// TIA Portal V17 export
// export: Created 2023-02-14T02:49:47.3102049Z, ExportSetting WithDefaults, DisplayName Totally Integrated Automation Portal, DisplayVersion V17, DisplayName TIA Portal Openness, DisplayVersion V17, DisplayName TIA Portal Teamcenter Gateway, DisplayVersion V17, DisplayName TIA Portal Version Control Interface, DisplayVersion V17, DisplayName SINAMICS Startdrive Advanced, DisplayVersion V17, DisplayName SINAMICS Startdrive G130, G150, S120, S150, SINAMICS MV, S210, DisplayVersion V17, DisplayName SINAMICS Startdrive G110M, G120, G120C, G120D, G120P, G115D, DisplayVersion V17, DisplayName STEP 7 Professional, DisplayVersion V17, DisplayName STEP 7 Safety, DisplayVersion V17, DisplayName WinCC Professional, DisplayVersion V17
FUNCTION "Buffer" : Void   // FC11, LAD
{ S7_Optimized_Access := 'TRUE' }
VERSION : 0.1
// stored: AutoNumber true, IsIECCheckEnabled false, SetENOAutomatically false, UDAEnableTagReadback false
BEGIN

REGION Network 1: BFT 61 Rework 32
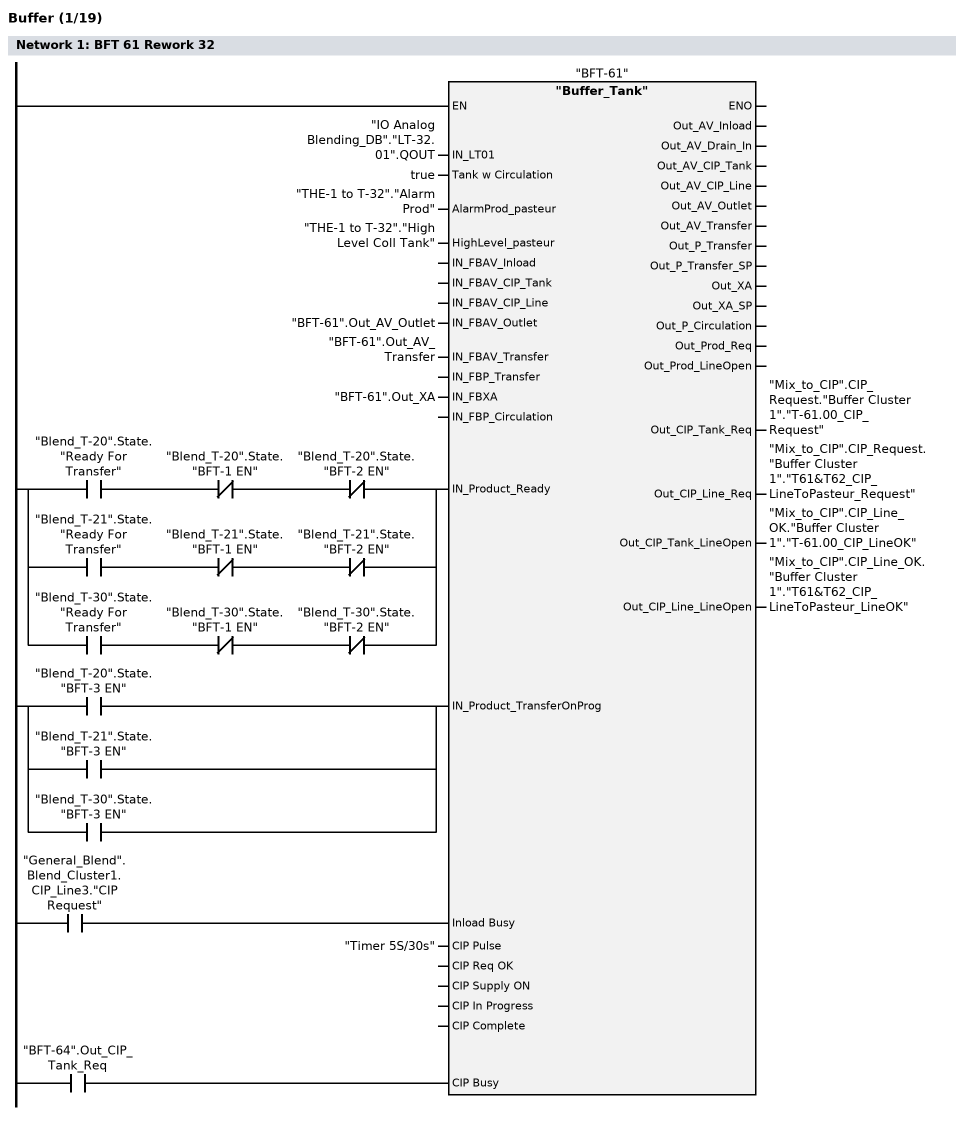
   RUNG wire#powerrail
      "BFT-61"(IN_Product_Ready := wire#w1, IN_Product_TransferOnProg := wire#w2, "Inload Busy" := wire#w3, "CIP Busy" := wire#w4, IN_LT01 := "IO Analog Blending_DB"."LT-32.01".QOUT, "Tank w Circulation" := true, AlarmProd_pasteur := "THE-1 to T-32"."Alarm Prod", HighLevel_pasteur := "THE-1 to T-32"."High Level Coll Tank", IN_FBAV_Inload :=, IN_FBAV_CIP_Tank :=, IN_FBAV_CIP_Line :=, IN_FBAV_Outlet := "BFT-61".Out_AV_Outlet, IN_FBAV_Transfer := "BFT-61".Out_AV_Transfer, IN_FBP_Transfer :=, IN_FBXA := "BFT-61".Out_XA, IN_FBP_Circulation :=, "CIP Pulse" := "Timer 5S/30s", "CIP Req OK" :=, "CIP Supply ON" :=, "CIP In Progress" :=, "CIP Complete" :=, Out_AV_Inload =>, Out_AV_Drain_In =>, Out_AV_CIP_Tank =>, Out_AV_CIP_Line =>, Out_AV_Outlet =>, Out_AV_Transfer =>, Out_P_Transfer =>, Out_P_Transfer_SP =>, Out_XA =>, Out_XA_SP =>, Out_P_Circulation =>, Out_Prod_Req =>, Out_Prod_LineOpen =>, Out_CIP_Tank_Req => "Mix_to_CIP".CIP_Request."Buffer Cluster 1"."T-61.00_CIP_Request", Out_CIP_Line_Req => "Mix_to_CIP".CIP_Request."Buffer Cluster 1"."T61&T62_CIP_LineToPasteur_Request", Out_CIP_Tank_LineOpen => "Mix_to_CIP".CIP_Line_OK."Buffer Cluster 1"."T-61.00_CIP_LineOK", Out_CIP_Line_LineOpen => "Mix_to_CIP".CIP_Line_OK."Buffer Cluster 1"."T61&T62_CIP_LineToPasteur_LineOK")
   END_RUNG
   RUNG wire#powerrail
      Contact( "Blend_T-20".State."Ready For Transfer" )
      I_Contact( "Blend_T-20".State."BFT-1 EN" )
      I_Contact( "Blend_T-20".State."BFT-2 EN" )
   END_RUNG wire#w1
   RUNG wire#powerrail
      Contact( "Blend_T-21".State."Ready For Transfer" )
      I_Contact( "Blend_T-21".State."BFT-1 EN" )
      I_Contact( "Blend_T-21".State."BFT-2 EN" )
   END_RUNG wire#w1
   RUNG wire#powerrail
      Contact( "Blend_T-30".State."Ready For Transfer" )
      I_Contact( "Blend_T-30".State."BFT-1 EN" )
      I_Contact( "Blend_T-30".State."BFT-2 EN" )
   END_RUNG wire#w1
   RUNG wire#powerrail
      Contact( "Blend_T-20".State."BFT-3 EN" )
   END_RUNG wire#w2
   RUNG wire#powerrail
      Contact( "Blend_T-21".State."BFT-3 EN" )
   END_RUNG wire#w2
   RUNG wire#powerrail
      Contact( "Blend_T-30".State."BFT-3 EN" )
   END_RUNG wire#w2
   RUNG wire#powerrail
      Contact( "General_Blend".Blend_Cluster1.CIP_Line3."CIP Request" )
   END_RUNG wire#w3
   RUNG wire#powerrail
      Contact( "BFT-64".Out_CIP_Tank_Req )
   END_RUNG wire#w4
   // the same network as SCL:
   "BFT-61"(IN_LT01 := "IO Analog Blending_DB"."LT-32.01".QOUT,   // "Buffer_Tank"
            "Tank w Circulation" := true,
            AlarmProd_pasteur := "THE-1 to T-32"."Alarm Prod",
            HighLevel_pasteur := "THE-1 to T-32"."High Level Coll Tank",
            IN_FBAV_Outlet := "BFT-61".Out_AV_Outlet,
            IN_FBAV_Transfer := "BFT-61".Out_AV_Transfer,
            IN_FBXA := "BFT-61".Out_XA,
            IN_Product_Ready := ("Blend_T-20".State."Ready For Transfer" AND NOT "Blend_T-20".State."BFT-1 EN" AND NOT "Blend_T-20".State."BFT-2 EN") OR ("Blend_T-21".State."Ready For Transfer" AND NOT "Blend_T-21".State."BFT-1 EN" AND NOT "Blend_T-21".State."BFT-2 EN") OR ("Blend_T-30".State."Ready For Transfer" AND NOT "Blend_T-30".State."BFT-1 EN" AND NOT "Blend_T-30".State."BFT-2 EN"),
            IN_Product_TransferOnProg := "Blend_T-20".State."BFT-3 EN" OR "Blend_T-21".State."BFT-3 EN" OR "Blend_T-30".State."BFT-3 EN",
            "Inload Busy" := "General_Blend".Blend_Cluster1.CIP_Line3."CIP Request",
            "CIP Pulse" := "Timer 5S/30s",
            "CIP Busy" := "BFT-64".Out_CIP_Tank_Req,
            Out_CIP_Tank_Req => "Mix_to_CIP".CIP_Request."Buffer Cluster 1"."T-61.00_CIP_Request",
            Out_CIP_Line_Req => "Mix_to_CIP".CIP_Request."Buffer Cluster 1"."T61&T62_CIP_LineToPasteur_Request",
            Out_CIP_Tank_LineOpen => "Mix_to_CIP".CIP_Line_OK."Buffer Cluster 1"."T-61.00_CIP_LineOK",
            Out_CIP_Line_LineOpen => "Mix_to_CIP".CIP_Line_OK."Buffer Cluster 1"."T61&T62_CIP_LineToPasteur_LineOK");
END_REGION

REGION Network 2: BFT 61 Feedback Instrument
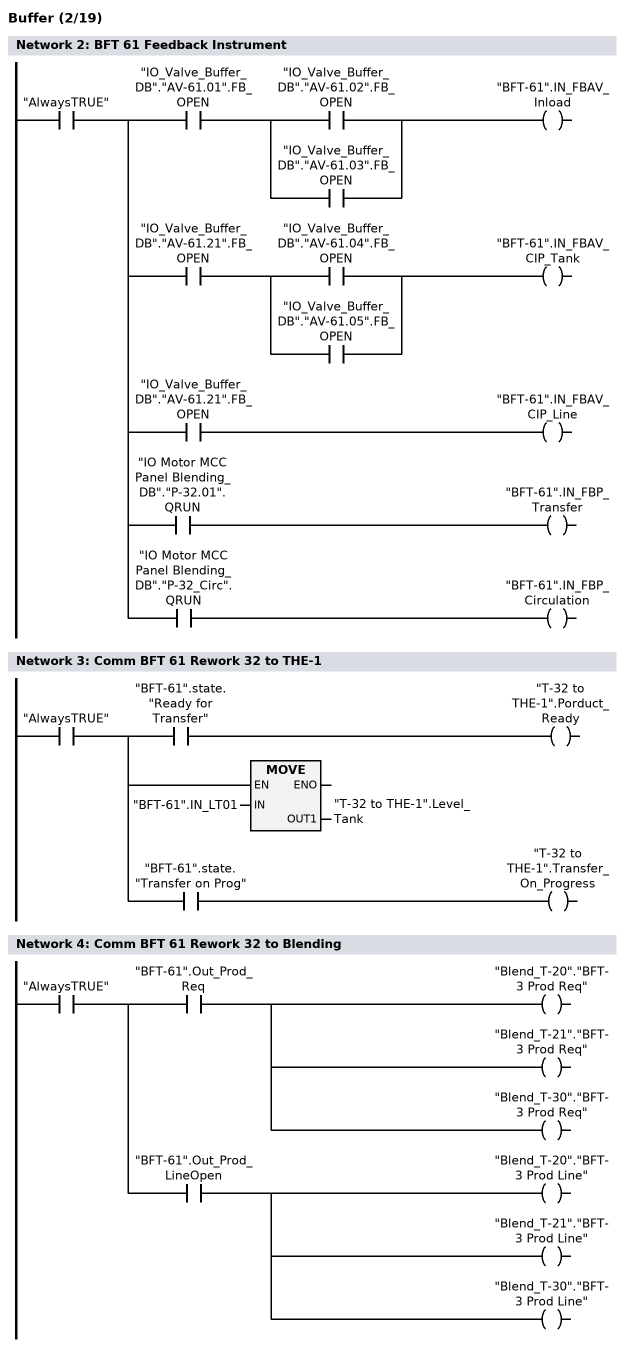
   RUNG wire#powerrail
      Contact( "AlwaysTRUE" )
      wire#w1
      Contact( "IO_Valve_Buffer_DB"."AV-61.01".FB_OPEN )
      wire#w2
      Contact( "IO_Valve_Buffer_DB"."AV-61.02".FB_OPEN )
      wire#w3
      Coil( "BFT-61".IN_FBAV_Inload )
   END_RUNG
   RUNG wire#w2
      Contact( "IO_Valve_Buffer_DB"."AV-61.03".FB_OPEN )
   END_RUNG wire#w3
   RUNG wire#w1
      Contact( "IO_Valve_Buffer_DB"."AV-61.21".FB_OPEN )
      wire#w4
      Contact( "IO_Valve_Buffer_DB"."AV-61.04".FB_OPEN )
      wire#w5
      Coil( "BFT-61".IN_FBAV_CIP_Tank )
   END_RUNG
   RUNG wire#w4
      Contact( "IO_Valve_Buffer_DB"."AV-61.05".FB_OPEN )
   END_RUNG wire#w5
   RUNG wire#w1
      Contact( "IO_Valve_Buffer_DB"."AV-61.21".FB_OPEN )
      Coil( "BFT-61".IN_FBAV_CIP_Line )
   END_RUNG
   RUNG wire#w1
      Contact( "IO Motor MCC Panel Blending_DB"."P-32.01".QRUN )
      Coil( "BFT-61".IN_FBP_Transfer )
   END_RUNG
   RUNG wire#w1
      Contact( "IO Motor MCC Panel Blending_DB"."P-32_Circ".QRUN )
      Coil( "BFT-61".IN_FBP_Circulation )
   END_RUNG
   // the same network as SCL:
   "BFT-61".IN_FBAV_Inload := "AlwaysTRUE" AND "IO_Valve_Buffer_DB"."AV-61.01".FB_OPEN AND ("IO_Valve_Buffer_DB"."AV-61.02".FB_OPEN OR "IO_Valve_Buffer_DB"."AV-61.03".FB_OPEN);
   "BFT-61".IN_FBAV_CIP_Tank := "AlwaysTRUE" AND "IO_Valve_Buffer_DB"."AV-61.21".FB_OPEN AND ("IO_Valve_Buffer_DB"."AV-61.04".FB_OPEN OR "IO_Valve_Buffer_DB"."AV-61.05".FB_OPEN);
   "BFT-61".IN_FBAV_CIP_Line := "AlwaysTRUE" AND "IO_Valve_Buffer_DB"."AV-61.21".FB_OPEN;
   "BFT-61".IN_FBP_Transfer := "AlwaysTRUE" AND "IO Motor MCC Panel Blending_DB"."P-32.01".QRUN;
   "BFT-61".IN_FBP_Circulation := "AlwaysTRUE" AND "IO Motor MCC Panel Blending_DB"."P-32_Circ".QRUN;
END_REGION

REGION Network 3: Comm BFT 61 Rework 32 to THE-1
   RUNG wire#powerrail
      Contact( "AlwaysTRUE" )
      wire#w1
      Contact( "BFT-61".state."Ready for Transfer" )
      Coil( "T-32 to THE-1".Porduct_Ready )
   END_RUNG
   RUNG wire#w1
      Move(in := "BFT-61".IN_LT01, out1 => "T-32 to THE-1".Level_Tank)
   END_RUNG
   RUNG wire#w1
      Contact( "BFT-61".state."Transfer on Prog" )
      Coil( "T-32 to THE-1".Transfer_On_Progress )
   END_RUNG
   // the same network as SCL:
   "T-32 to THE-1".Porduct_Ready := "AlwaysTRUE" AND "BFT-61".state."Ready for Transfer";
   IF "AlwaysTRUE" THEN "T-32 to THE-1".Level_Tank := "BFT-61".IN_LT01; END_IF;
   "T-32 to THE-1".Transfer_On_Progress := "AlwaysTRUE" AND "BFT-61".state."Transfer on Prog";
END_REGION

REGION Network 4: Comm BFT 61 Rework 32 to Blending
   RUNG wire#powerrail
      Contact( "AlwaysTRUE" )
      wire#w1
      Contact( "BFT-61".Out_Prod_Req )
      wire#w2
      Coil( "Blend_T-20"."BFT-3 Prod Req" )
   END_RUNG
   RUNG wire#w2
      Coil( "Blend_T-21"."BFT-3 Prod Req" )
   END_RUNG
   RUNG wire#w2
      Coil( "Blend_T-30"."BFT-3 Prod Req" )
   END_RUNG
   RUNG wire#w1
      Contact( "BFT-61".Out_Prod_LineOpen )
      wire#w3
      Coil( "Blend_T-20"."BFT-3 Prod Line" )
   END_RUNG
   RUNG wire#w3
      Coil( "Blend_T-21"."BFT-3 Prod Line" )
   END_RUNG
   RUNG wire#w3
      Coil( "Blend_T-30"."BFT-3 Prod Line" )
   END_RUNG
   // the same network as SCL:
   "Blend_T-20"."BFT-3 Prod Req" := "AlwaysTRUE" AND "BFT-61".Out_Prod_Req;
   "Blend_T-21"."BFT-3 Prod Req" := "Blend_T-20"."BFT-3 Prod Req";
   "Blend_T-30"."BFT-3 Prod Req" := "Blend_T-20"."BFT-3 Prod Req";
   "Blend_T-20"."BFT-3 Prod Line" := "AlwaysTRUE" AND "BFT-61".Out_Prod_LineOpen;
   "Blend_T-21"."BFT-3 Prod Line" := "Blend_T-20"."BFT-3 Prod Line";
   "Blend_T-30"."BFT-3 Prod Line" := "Blend_T-20"."BFT-3 Prod Line";
END_REGION

REGION Network 6: BFT 64 Rework 22
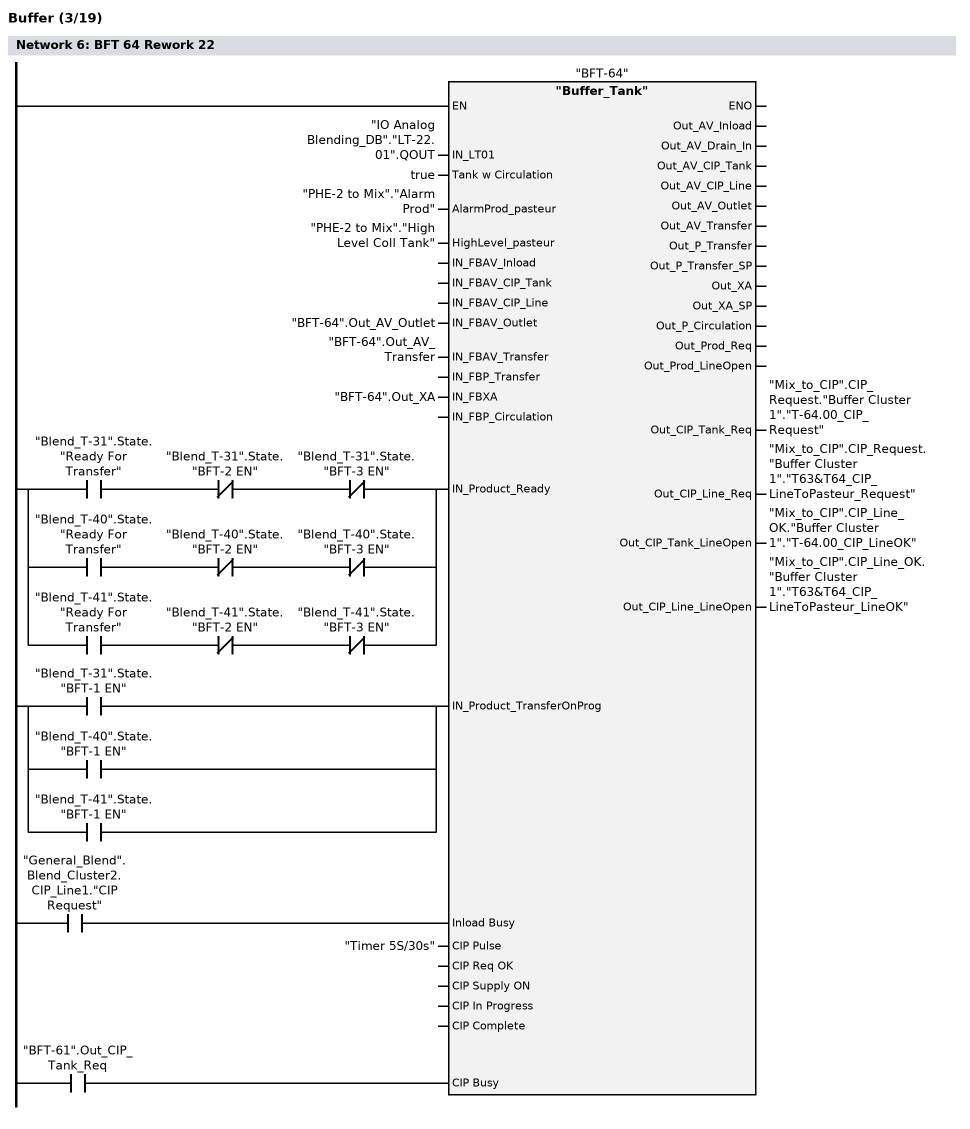
   RUNG wire#powerrail
      "BFT-64"(IN_Product_Ready := wire#w1, IN_Product_TransferOnProg := wire#w2, "Inload Busy" := wire#w3, "CIP Busy" := wire#w4, IN_LT01 := "IO Analog Blending_DB"."LT-22.01".QOUT, "Tank w Circulation" := true, AlarmProd_pasteur := "PHE-2 to Mix"."Alarm Prod", HighLevel_pasteur := "PHE-2 to Mix"."High Level Coll Tank", IN_FBAV_Inload :=, IN_FBAV_CIP_Tank :=, IN_FBAV_CIP_Line :=, IN_FBAV_Outlet := "BFT-64".Out_AV_Outlet, IN_FBAV_Transfer := "BFT-64".Out_AV_Transfer, IN_FBP_Transfer :=, IN_FBXA := "BFT-64".Out_XA, IN_FBP_Circulation :=, "CIP Pulse" := "Timer 5S/30s", "CIP Req OK" :=, "CIP Supply ON" :=, "CIP In Progress" :=, "CIP Complete" :=, Out_AV_Inload =>, Out_AV_Drain_In =>, Out_AV_CIP_Tank =>, Out_AV_CIP_Line =>, Out_AV_Outlet =>, Out_AV_Transfer =>, Out_P_Transfer =>, Out_P_Transfer_SP =>, Out_XA =>, Out_XA_SP =>, Out_P_Circulation =>, Out_Prod_Req =>, Out_Prod_LineOpen =>, Out_CIP_Tank_Req => "Mix_to_CIP".CIP_Request."Buffer Cluster 1"."T-64.00_CIP_Request", Out_CIP_Line_Req => "Mix_to_CIP".CIP_Request."Buffer Cluster 1"."T63&T64_CIP_LineToPasteur_Request", Out_CIP_Tank_LineOpen => "Mix_to_CIP".CIP_Line_OK."Buffer Cluster 1"."T-64.00_CIP_LineOK", Out_CIP_Line_LineOpen => "Mix_to_CIP".CIP_Line_OK."Buffer Cluster 1"."T63&T64_CIP_LineToPasteur_LineOK")
   END_RUNG
   RUNG wire#powerrail
      Contact( "Blend_T-31".State."Ready For Transfer" )
      I_Contact( "Blend_T-31".State."BFT-2 EN" )
      I_Contact( "Blend_T-31".State."BFT-3 EN" )
   END_RUNG wire#w1
   RUNG wire#powerrail
      Contact( "Blend_T-40".State."Ready For Transfer" )
      I_Contact( "Blend_T-40".State."BFT-2 EN" )
      I_Contact( "Blend_T-40".State."BFT-3 EN" )
   END_RUNG wire#w1
   RUNG wire#powerrail
      Contact( "Blend_T-41".State."Ready For Transfer" )
      I_Contact( "Blend_T-41".State."BFT-2 EN" )
      I_Contact( "Blend_T-41".State."BFT-3 EN" )
   END_RUNG wire#w1
   RUNG wire#powerrail
      Contact( "Blend_T-31".State."BFT-1 EN" )
   END_RUNG wire#w2
   RUNG wire#powerrail
      Contact( "Blend_T-40".State."BFT-1 EN" )
   END_RUNG wire#w2
   RUNG wire#powerrail
      Contact( "Blend_T-41".State."BFT-1 EN" )
   END_RUNG wire#w2
   RUNG wire#powerrail
      Contact( "General_Blend".Blend_Cluster2.CIP_Line1."CIP Request" )
   END_RUNG wire#w3
   RUNG wire#powerrail
      Contact( "BFT-61".Out_CIP_Tank_Req )
   END_RUNG wire#w4
   // the same network as SCL:
   "BFT-64"(IN_LT01 := "IO Analog Blending_DB"."LT-22.01".QOUT,   // "Buffer_Tank"
            "Tank w Circulation" := true,
            AlarmProd_pasteur := "PHE-2 to Mix"."Alarm Prod",
            HighLevel_pasteur := "PHE-2 to Mix"."High Level Coll Tank",
            IN_FBAV_Outlet := "BFT-64".Out_AV_Outlet,
            IN_FBAV_Transfer := "BFT-64".Out_AV_Transfer,
            IN_FBXA := "BFT-64".Out_XA,
            IN_Product_Ready := ("Blend_T-31".State."Ready For Transfer" AND NOT "Blend_T-31".State."BFT-2 EN" AND NOT "Blend_T-31".State."BFT-3 EN") OR ("Blend_T-40".State."Ready For Transfer" AND NOT "Blend_T-40".State."BFT-2 EN" AND NOT "Blend_T-40".State."BFT-3 EN") OR ("Blend_T-41".State."Ready For Transfer" AND NOT "Blend_T-41".State."BFT-2 EN" AND NOT "Blend_T-41".State."BFT-3 EN"),
            IN_Product_TransferOnProg := "Blend_T-31".State."BFT-1 EN" OR "Blend_T-40".State."BFT-1 EN" OR "Blend_T-41".State."BFT-1 EN",
            "Inload Busy" := "General_Blend".Blend_Cluster2.CIP_Line1."CIP Request",
            "CIP Pulse" := "Timer 5S/30s",
            "CIP Busy" := "BFT-61".Out_CIP_Tank_Req,
            Out_CIP_Tank_Req => "Mix_to_CIP".CIP_Request."Buffer Cluster 1"."T-64.00_CIP_Request",
            Out_CIP_Line_Req => "Mix_to_CIP".CIP_Request."Buffer Cluster 1"."T63&T64_CIP_LineToPasteur_Request",
            Out_CIP_Tank_LineOpen => "Mix_to_CIP".CIP_Line_OK."Buffer Cluster 1"."T-64.00_CIP_LineOK",
            Out_CIP_Line_LineOpen => "Mix_to_CIP".CIP_Line_OK."Buffer Cluster 1"."T63&T64_CIP_LineToPasteur_LineOK");
END_REGION

REGION Network 7: BFT 64 Feedback Instrument
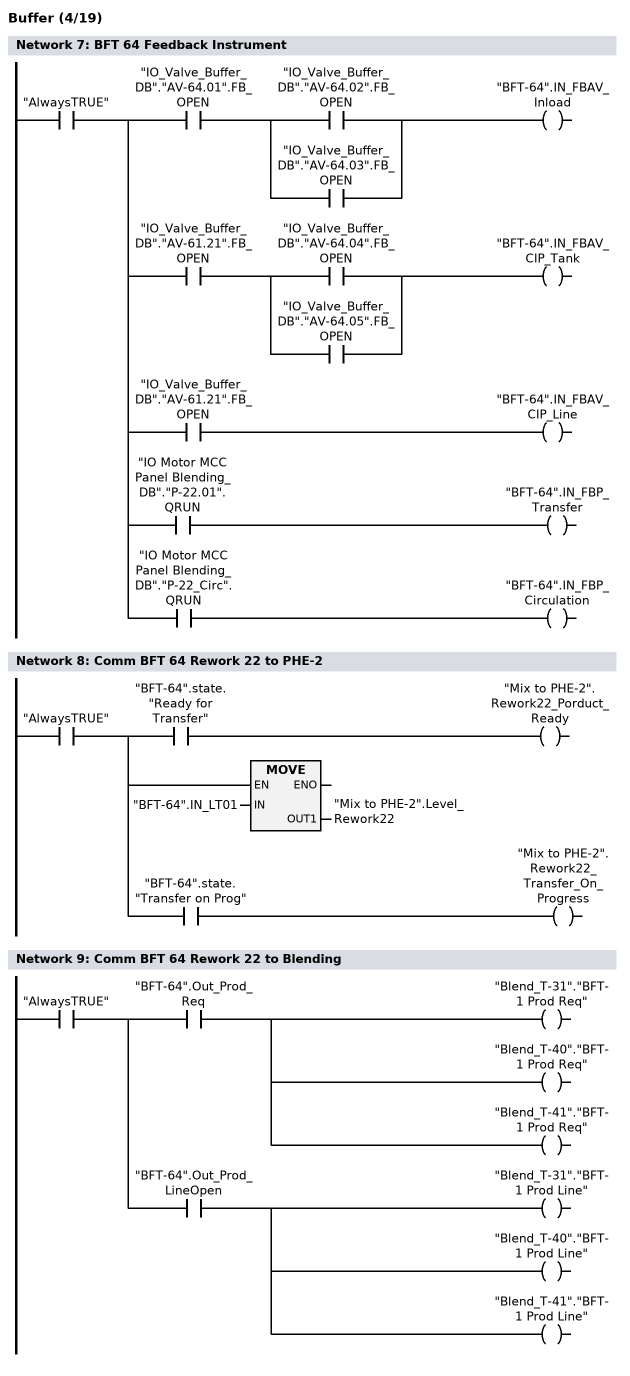
   RUNG wire#powerrail
      Contact( "AlwaysTRUE" )
      wire#w1
      Contact( "IO_Valve_Buffer_DB"."AV-64.01".FB_OPEN )
      wire#w2
      Contact( "IO_Valve_Buffer_DB"."AV-64.02".FB_OPEN )
      wire#w3
      Coil( "BFT-64".IN_FBAV_Inload )
   END_RUNG
   RUNG wire#w2
      Contact( "IO_Valve_Buffer_DB"."AV-64.03".FB_OPEN )
   END_RUNG wire#w3
   RUNG wire#w1
      Contact( "IO_Valve_Buffer_DB"."AV-61.21".FB_OPEN )
      wire#w4
      Contact( "IO_Valve_Buffer_DB"."AV-64.04".FB_OPEN )
      wire#w5
      Coil( "BFT-64".IN_FBAV_CIP_Tank )
   END_RUNG
   RUNG wire#w4
      Contact( "IO_Valve_Buffer_DB"."AV-64.05".FB_OPEN )
   END_RUNG wire#w5
   RUNG wire#w1
      Contact( "IO_Valve_Buffer_DB"."AV-61.21".FB_OPEN )
      Coil( "BFT-64".IN_FBAV_CIP_Line )
   END_RUNG
   RUNG wire#w1
      Contact( "IO Motor MCC Panel Blending_DB"."P-22.01".QRUN )
      Coil( "BFT-64".IN_FBP_Transfer )
   END_RUNG
   RUNG wire#w1
      Contact( "IO Motor MCC Panel Blending_DB"."P-22_Circ".QRUN )
      Coil( "BFT-64".IN_FBP_Circulation )
   END_RUNG
   // the same network as SCL:
   "BFT-64".IN_FBAV_Inload := "AlwaysTRUE" AND "IO_Valve_Buffer_DB"."AV-64.01".FB_OPEN AND ("IO_Valve_Buffer_DB"."AV-64.02".FB_OPEN OR "IO_Valve_Buffer_DB"."AV-64.03".FB_OPEN);
   "BFT-64".IN_FBAV_CIP_Tank := "AlwaysTRUE" AND "IO_Valve_Buffer_DB"."AV-61.21".FB_OPEN AND ("IO_Valve_Buffer_DB"."AV-64.04".FB_OPEN OR "IO_Valve_Buffer_DB"."AV-64.05".FB_OPEN);
   "BFT-64".IN_FBAV_CIP_Line := "AlwaysTRUE" AND "IO_Valve_Buffer_DB"."AV-61.21".FB_OPEN;
   "BFT-64".IN_FBP_Transfer := "AlwaysTRUE" AND "IO Motor MCC Panel Blending_DB"."P-22.01".QRUN;
   "BFT-64".IN_FBP_Circulation := "AlwaysTRUE" AND "IO Motor MCC Panel Blending_DB"."P-22_Circ".QRUN;
END_REGION

REGION Network 8: Comm BFT 64 Rework 22 to PHE-2
   RUNG wire#powerrail
      Contact( "AlwaysTRUE" )
      wire#w1
      Contact( "BFT-64".state."Ready for Transfer" )
      Coil( "Mix to PHE-2".Rework22_Porduct_Ready )
   END_RUNG
   RUNG wire#w1
      Move(in := "BFT-64".IN_LT01, out1 => "Mix to PHE-2".Level_Rework22)
   END_RUNG
   RUNG wire#w1
      Contact( "BFT-64".state."Transfer on Prog" )
      Coil( "Mix to PHE-2".Rework22_Transfer_On_Progress )
   END_RUNG
   // the same network as SCL:
   "Mix to PHE-2".Rework22_Porduct_Ready := "AlwaysTRUE" AND "BFT-64".state."Ready for Transfer";
   IF "AlwaysTRUE" THEN "Mix to PHE-2".Level_Rework22 := "BFT-64".IN_LT01; END_IF;
   "Mix to PHE-2".Rework22_Transfer_On_Progress := "AlwaysTRUE" AND "BFT-64".state."Transfer on Prog";
END_REGION

REGION Network 9: Comm BFT 64 Rework 22 to Blending
   RUNG wire#powerrail
      Contact( "AlwaysTRUE" )
      wire#w1
      Contact( "BFT-64".Out_Prod_Req )
      wire#w2
      Coil( "Blend_T-31"."BFT-1 Prod Req" )
   END_RUNG
   RUNG wire#w2
      Coil( "Blend_T-40"."BFT-1 Prod Req" )
   END_RUNG
   RUNG wire#w2
      Coil( "Blend_T-41"."BFT-1 Prod Req" )
   END_RUNG
   RUNG wire#w1
      Contact( "BFT-64".Out_Prod_LineOpen )
      wire#w3
      Coil( "Blend_T-31"."BFT-1 Prod Line" )
   END_RUNG
   RUNG wire#w3
      Coil( "Blend_T-40"."BFT-1 Prod Line" )
   END_RUNG
   RUNG wire#w3
      Coil( "Blend_T-41"."BFT-1 Prod Line" )
   END_RUNG
   // the same network as SCL:
   "Blend_T-31"."BFT-1 Prod Req" := "AlwaysTRUE" AND "BFT-64".Out_Prod_Req;
   "Blend_T-40"."BFT-1 Prod Req" := "Blend_T-31"."BFT-1 Prod Req";
   "Blend_T-41"."BFT-1 Prod Req" := "Blend_T-31"."BFT-1 Prod Req";
   "Blend_T-31"."BFT-1 Prod Line" := "AlwaysTRUE" AND "BFT-64".Out_Prod_LineOpen;
   "Blend_T-40"."BFT-1 Prod Line" := "Blend_T-31"."BFT-1 Prod Line";
   "Blend_T-41"."BFT-1 Prod Line" := "Blend_T-31"."BFT-1 Prod Line";
END_REGION

REGION Network 11: BFT 65
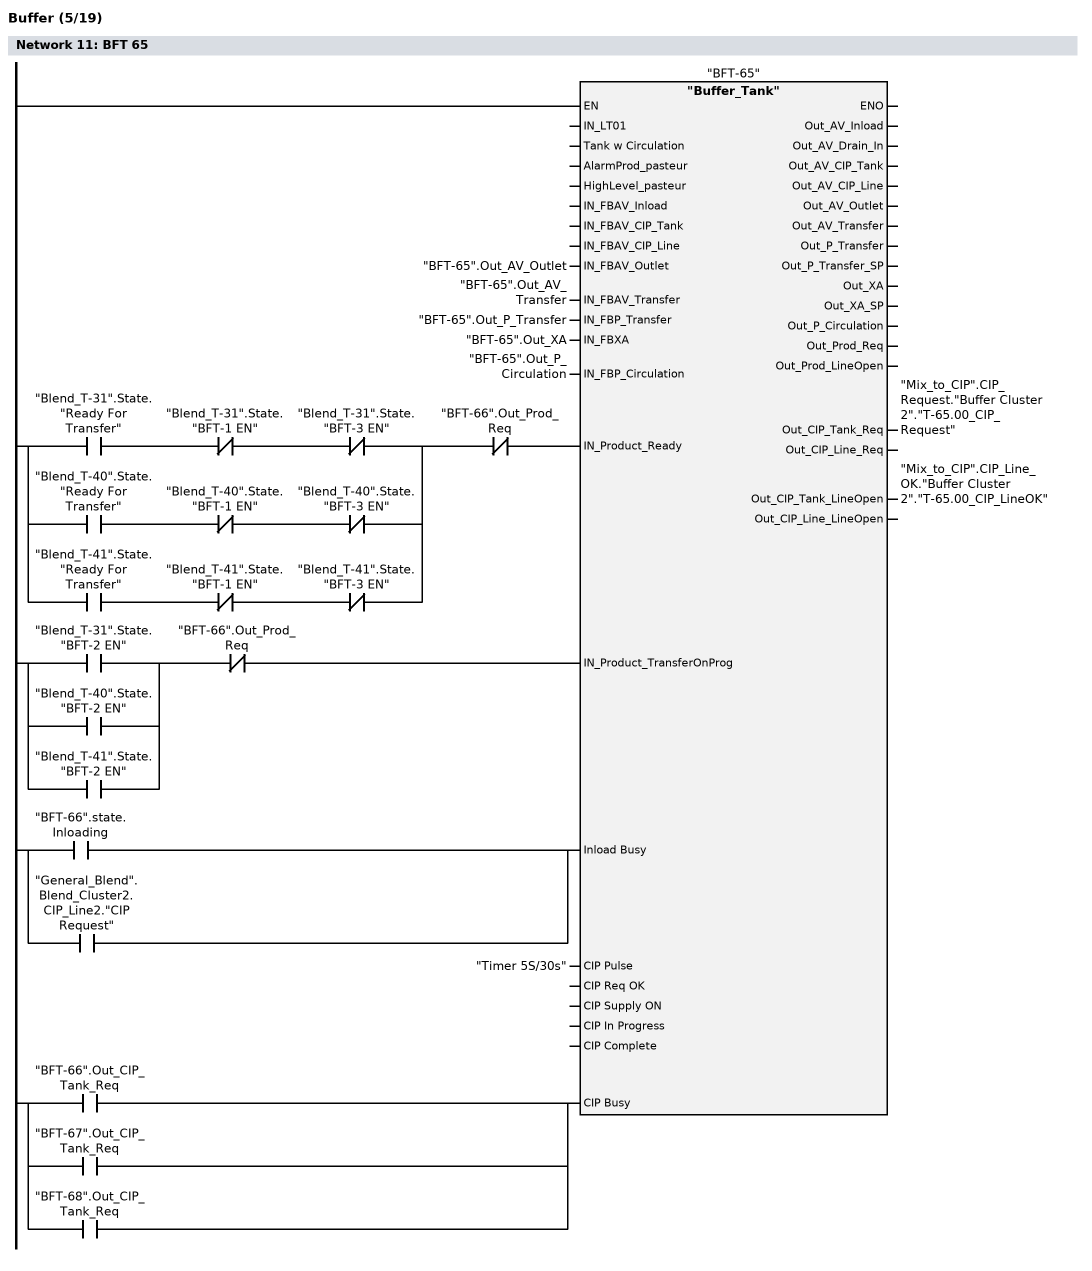
   RUNG wire#powerrail
      "BFT-65"(IN_Product_Ready := wire#w2, IN_Product_TransferOnProg := wire#w4, "Inload Busy" := wire#w5, "CIP Busy" := wire#w6, IN_LT01 :=, "Tank w Circulation" :=, AlarmProd_pasteur :=, HighLevel_pasteur :=, IN_FBAV_Inload :=, IN_FBAV_CIP_Tank :=, IN_FBAV_CIP_Line :=, IN_FBAV_Outlet := "BFT-65".Out_AV_Outlet, IN_FBAV_Transfer := "BFT-65".Out_AV_Transfer, IN_FBP_Transfer := "BFT-65".Out_P_Transfer, IN_FBXA := "BFT-65".Out_XA, IN_FBP_Circulation := "BFT-65".Out_P_Circulation, "CIP Pulse" := "Timer 5S/30s", "CIP Req OK" :=, "CIP Supply ON" :=, "CIP In Progress" :=, "CIP Complete" :=, Out_AV_Inload =>, Out_AV_Drain_In =>, Out_AV_CIP_Tank =>, Out_AV_CIP_Line =>, Out_AV_Outlet =>, Out_AV_Transfer =>, Out_P_Transfer =>, Out_P_Transfer_SP =>, Out_XA =>, Out_XA_SP =>, Out_P_Circulation =>, Out_Prod_Req =>, Out_Prod_LineOpen =>, Out_CIP_Tank_Req => "Mix_to_CIP".CIP_Request."Buffer Cluster 2"."T-65.00_CIP_Request", Out_CIP_Line_Req =>, Out_CIP_Tank_LineOpen => "Mix_to_CIP".CIP_Line_OK."Buffer Cluster 2"."T-65.00_CIP_LineOK", Out_CIP_Line_LineOpen =>)
   END_RUNG
   RUNG wire#powerrail
      Contact( "Blend_T-31".State."Ready For Transfer" )
      I_Contact( "Blend_T-31".State."BFT-1 EN" )
      I_Contact( "Blend_T-31".State."BFT-3 EN" )
      wire#w1
      I_Contact( "BFT-66".Out_Prod_Req )
   END_RUNG wire#w2
   RUNG wire#powerrail
      Contact( "Blend_T-40".State."Ready For Transfer" )
      I_Contact( "Blend_T-40".State."BFT-1 EN" )
      I_Contact( "Blend_T-40".State."BFT-3 EN" )
   END_RUNG wire#w1
   RUNG wire#powerrail
      Contact( "Blend_T-41".State."Ready For Transfer" )
      I_Contact( "Blend_T-41".State."BFT-1 EN" )
      I_Contact( "Blend_T-41".State."BFT-3 EN" )
   END_RUNG wire#w1
   RUNG wire#powerrail
      Contact( "Blend_T-31".State."BFT-2 EN" )
      wire#w3
      I_Contact( "BFT-66".Out_Prod_Req )
   END_RUNG wire#w4
   RUNG wire#powerrail
      Contact( "Blend_T-40".State."BFT-2 EN" )
   END_RUNG wire#w3
   RUNG wire#powerrail
      Contact( "Blend_T-41".State."BFT-2 EN" )
   END_RUNG wire#w3
   RUNG wire#powerrail
      Contact( "BFT-66".state.Inloading )
   END_RUNG wire#w5
   RUNG wire#powerrail
      Contact( "General_Blend".Blend_Cluster2.CIP_Line2."CIP Request" )
   END_RUNG wire#w5
   RUNG wire#powerrail
      Contact( "BFT-66".Out_CIP_Tank_Req )
   END_RUNG wire#w6
   RUNG wire#powerrail
      Contact( "BFT-67".Out_CIP_Tank_Req )
   END_RUNG wire#w6
   RUNG wire#powerrail
      Contact( "BFT-68".Out_CIP_Tank_Req )
   END_RUNG wire#w6
   // the same network as SCL:
   "BFT-65"(IN_FBAV_Outlet := "BFT-65".Out_AV_Outlet,   // "Buffer_Tank"
            IN_FBAV_Transfer := "BFT-65".Out_AV_Transfer,
            IN_FBP_Transfer := "BFT-65".Out_P_Transfer,
            IN_FBXA := "BFT-65".Out_XA,
            IN_FBP_Circulation := "BFT-65".Out_P_Circulation,
            IN_Product_Ready := (("Blend_T-31".State."Ready For Transfer" AND NOT "Blend_T-31".State."BFT-1 EN" AND NOT "Blend_T-31".State."BFT-3 EN") OR ("Blend_T-40".State."Ready For Transfer" AND NOT "Blend_T-40".State."BFT-1 EN" AND NOT "Blend_T-40".State."BFT-3 EN") OR ("Blend_T-41".State."Ready For Transfer" AND NOT "Blend_T-41".State."BFT-1 EN" AND NOT "Blend_T-41".State."BFT-3 EN")) AND NOT "BFT-66".Out_Prod_Req,
            IN_Product_TransferOnProg := ("Blend_T-31".State."BFT-2 EN" OR "Blend_T-40".State."BFT-2 EN" OR "Blend_T-41".State."BFT-2 EN") AND NOT "BFT-66".Out_Prod_Req,
            "Inload Busy" := "BFT-66".state.Inloading OR "General_Blend".Blend_Cluster2.CIP_Line2."CIP Request",
            "CIP Pulse" := "Timer 5S/30s",
            "CIP Busy" := "BFT-66".Out_CIP_Tank_Req OR "BFT-67".Out_CIP_Tank_Req OR "BFT-68".Out_CIP_Tank_Req,
            Out_CIP_Tank_Req => "Mix_to_CIP".CIP_Request."Buffer Cluster 2"."T-65.00_CIP_Request",
            Out_CIP_Tank_LineOpen => "Mix_to_CIP".CIP_Line_OK."Buffer Cluster 2"."T-65.00_CIP_LineOK");
END_REGION

REGION Network 12: BFT 65 Feedback Instrument
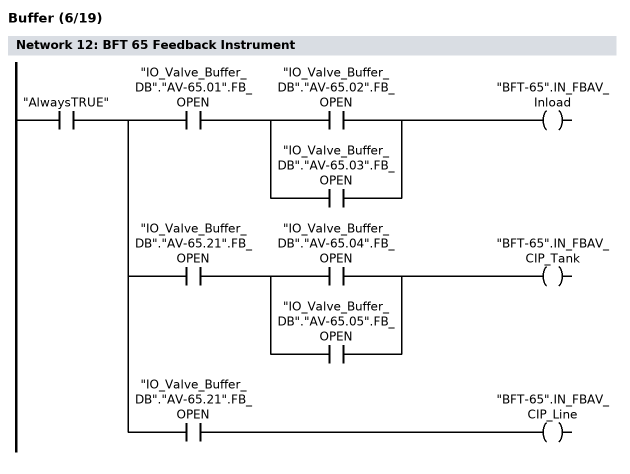
   RUNG wire#powerrail
      Contact( "AlwaysTRUE" )
      wire#w1
      Contact( "IO_Valve_Buffer_DB"."AV-65.01".FB_OPEN )
      wire#w2
      Contact( "IO_Valve_Buffer_DB"."AV-65.02".FB_OPEN )
      wire#w3
      Coil( "BFT-65".IN_FBAV_Inload )
   END_RUNG
   RUNG wire#w2
      Contact( "IO_Valve_Buffer_DB"."AV-65.03".FB_OPEN )
   END_RUNG wire#w3
   RUNG wire#w1
      Contact( "IO_Valve_Buffer_DB"."AV-65.21".FB_OPEN )
      wire#w4
      Contact( "IO_Valve_Buffer_DB"."AV-65.04".FB_OPEN )
      wire#w5
      Coil( "BFT-65".IN_FBAV_CIP_Tank )
   END_RUNG
   RUNG wire#w4
      Contact( "IO_Valve_Buffer_DB"."AV-65.05".FB_OPEN )
   END_RUNG wire#w5
   RUNG wire#w1
      Contact( "IO_Valve_Buffer_DB"."AV-65.21".FB_OPEN )
      Coil( "BFT-65".IN_FBAV_CIP_Line )
   END_RUNG
   // the same network as SCL:
   "BFT-65".IN_FBAV_Inload := "AlwaysTRUE" AND "IO_Valve_Buffer_DB"."AV-65.01".FB_OPEN AND ("IO_Valve_Buffer_DB"."AV-65.02".FB_OPEN OR "IO_Valve_Buffer_DB"."AV-65.03".FB_OPEN);
   "BFT-65".IN_FBAV_CIP_Tank := "AlwaysTRUE" AND "IO_Valve_Buffer_DB"."AV-65.21".FB_OPEN AND ("IO_Valve_Buffer_DB"."AV-65.04".FB_OPEN OR "IO_Valve_Buffer_DB"."AV-65.05".FB_OPEN);
   "BFT-65".IN_FBAV_CIP_Line := "AlwaysTRUE" AND "IO_Valve_Buffer_DB"."AV-65.21".FB_OPEN;
END_REGION

REGION Network 13: BFT 66
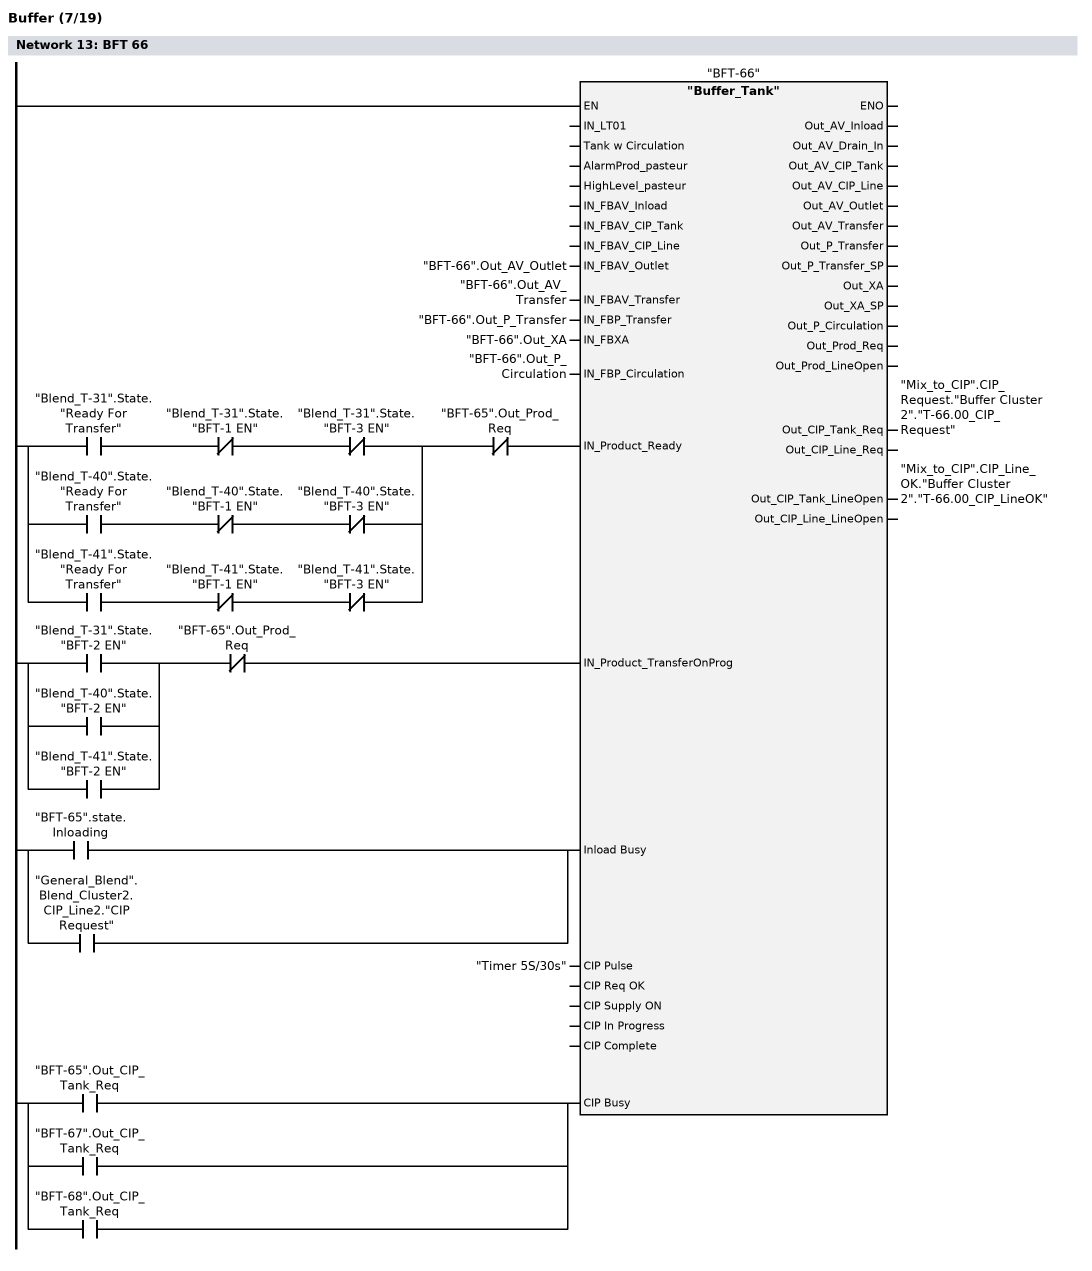
   RUNG wire#powerrail
      "BFT-66"(IN_Product_Ready := wire#w2, IN_Product_TransferOnProg := wire#w4, "Inload Busy" := wire#w5, "CIP Busy" := wire#w6, IN_LT01 :=, "Tank w Circulation" :=, AlarmProd_pasteur :=, HighLevel_pasteur :=, IN_FBAV_Inload :=, IN_FBAV_CIP_Tank :=, IN_FBAV_CIP_Line :=, IN_FBAV_Outlet := "BFT-66".Out_AV_Outlet, IN_FBAV_Transfer := "BFT-66".Out_AV_Transfer, IN_FBP_Transfer := "BFT-66".Out_P_Transfer, IN_FBXA := "BFT-66".Out_XA, IN_FBP_Circulation := "BFT-66".Out_P_Circulation, "CIP Pulse" := "Timer 5S/30s", "CIP Req OK" :=, "CIP Supply ON" :=, "CIP In Progress" :=, "CIP Complete" :=, Out_AV_Inload =>, Out_AV_Drain_In =>, Out_AV_CIP_Tank =>, Out_AV_CIP_Line =>, Out_AV_Outlet =>, Out_AV_Transfer =>, Out_P_Transfer =>, Out_P_Transfer_SP =>, Out_XA =>, Out_XA_SP =>, Out_P_Circulation =>, Out_Prod_Req =>, Out_Prod_LineOpen =>, Out_CIP_Tank_Req => "Mix_to_CIP".CIP_Request."Buffer Cluster 2"."T-66.00_CIP_Request", Out_CIP_Line_Req =>, Out_CIP_Tank_LineOpen => "Mix_to_CIP".CIP_Line_OK."Buffer Cluster 2"."T-66.00_CIP_LineOK", Out_CIP_Line_LineOpen =>)
   END_RUNG
   RUNG wire#powerrail
      Contact( "Blend_T-31".State."Ready For Transfer" )
      I_Contact( "Blend_T-31".State."BFT-1 EN" )
      I_Contact( "Blend_T-31".State."BFT-3 EN" )
      wire#w1
      I_Contact( "BFT-65".Out_Prod_Req )
   END_RUNG wire#w2
   RUNG wire#powerrail
      Contact( "Blend_T-40".State."Ready For Transfer" )
      I_Contact( "Blend_T-40".State."BFT-1 EN" )
      I_Contact( "Blend_T-40".State."BFT-3 EN" )
   END_RUNG wire#w1
   RUNG wire#powerrail
      Contact( "Blend_T-41".State."Ready For Transfer" )
      I_Contact( "Blend_T-41".State."BFT-1 EN" )
      I_Contact( "Blend_T-41".State."BFT-3 EN" )
   END_RUNG wire#w1
   RUNG wire#powerrail
      Contact( "Blend_T-31".State."BFT-2 EN" )
      wire#w3
      I_Contact( "BFT-65".Out_Prod_Req )
   END_RUNG wire#w4
   RUNG wire#powerrail
      Contact( "Blend_T-40".State."BFT-2 EN" )
   END_RUNG wire#w3
   RUNG wire#powerrail
      Contact( "Blend_T-41".State."BFT-2 EN" )
   END_RUNG wire#w3
   RUNG wire#powerrail
      Contact( "BFT-65".state.Inloading )
   END_RUNG wire#w5
   RUNG wire#powerrail
      Contact( "General_Blend".Blend_Cluster2.CIP_Line2."CIP Request" )
   END_RUNG wire#w5
   RUNG wire#powerrail
      Contact( "BFT-65".Out_CIP_Tank_Req )
   END_RUNG wire#w6
   RUNG wire#powerrail
      Contact( "BFT-67".Out_CIP_Tank_Req )
   END_RUNG wire#w6
   RUNG wire#powerrail
      Contact( "BFT-68".Out_CIP_Tank_Req )
   END_RUNG wire#w6
   // the same network as SCL:
   "BFT-66"(IN_FBAV_Outlet := "BFT-66".Out_AV_Outlet,   // "Buffer_Tank"
            IN_FBAV_Transfer := "BFT-66".Out_AV_Transfer,
            IN_FBP_Transfer := "BFT-66".Out_P_Transfer,
            IN_FBXA := "BFT-66".Out_XA,
            IN_FBP_Circulation := "BFT-66".Out_P_Circulation,
            IN_Product_Ready := (("Blend_T-31".State."Ready For Transfer" AND NOT "Blend_T-31".State."BFT-1 EN" AND NOT "Blend_T-31".State."BFT-3 EN") OR ("Blend_T-40".State."Ready For Transfer" AND NOT "Blend_T-40".State."BFT-1 EN" AND NOT "Blend_T-40".State."BFT-3 EN") OR ("Blend_T-41".State."Ready For Transfer" AND NOT "Blend_T-41".State."BFT-1 EN" AND NOT "Blend_T-41".State."BFT-3 EN")) AND NOT "BFT-65".Out_Prod_Req,
            IN_Product_TransferOnProg := ("Blend_T-31".State."BFT-2 EN" OR "Blend_T-40".State."BFT-2 EN" OR "Blend_T-41".State."BFT-2 EN") AND NOT "BFT-65".Out_Prod_Req,
            "Inload Busy" := "BFT-65".state.Inloading OR "General_Blend".Blend_Cluster2.CIP_Line2."CIP Request",
            "CIP Pulse" := "Timer 5S/30s",
            "CIP Busy" := "BFT-65".Out_CIP_Tank_Req OR "BFT-67".Out_CIP_Tank_Req OR "BFT-68".Out_CIP_Tank_Req,
            Out_CIP_Tank_Req => "Mix_to_CIP".CIP_Request."Buffer Cluster 2"."T-66.00_CIP_Request",
            Out_CIP_Tank_LineOpen => "Mix_to_CIP".CIP_Line_OK."Buffer Cluster 2"."T-66.00_CIP_LineOK");
END_REGION

REGION Network 14: BFT 66 Feedback Instrument
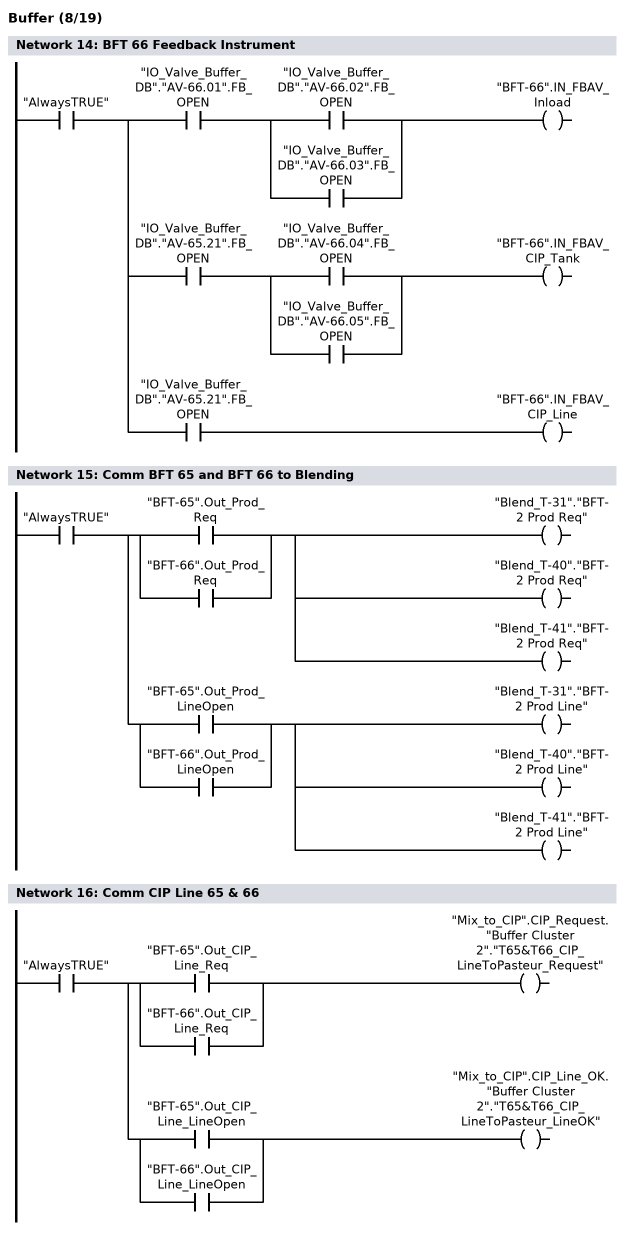
   RUNG wire#powerrail
      Contact( "AlwaysTRUE" )
      wire#w1
      Contact( "IO_Valve_Buffer_DB"."AV-66.01".FB_OPEN )
      wire#w2
      Contact( "IO_Valve_Buffer_DB"."AV-66.02".FB_OPEN )
      wire#w3
      Coil( "BFT-66".IN_FBAV_Inload )
   END_RUNG
   RUNG wire#w2
      Contact( "IO_Valve_Buffer_DB"."AV-66.03".FB_OPEN )
   END_RUNG wire#w3
   RUNG wire#w1
      Contact( "IO_Valve_Buffer_DB"."AV-65.21".FB_OPEN )
      wire#w4
      Contact( "IO_Valve_Buffer_DB"."AV-66.04".FB_OPEN )
      wire#w5
      Coil( "BFT-66".IN_FBAV_CIP_Tank )
   END_RUNG
   RUNG wire#w4
      Contact( "IO_Valve_Buffer_DB"."AV-66.05".FB_OPEN )
   END_RUNG wire#w5
   RUNG wire#w1
      Contact( "IO_Valve_Buffer_DB"."AV-65.21".FB_OPEN )
      Coil( "BFT-66".IN_FBAV_CIP_Line )
   END_RUNG
   // the same network as SCL:
   "BFT-66".IN_FBAV_Inload := "AlwaysTRUE" AND "IO_Valve_Buffer_DB"."AV-66.01".FB_OPEN AND ("IO_Valve_Buffer_DB"."AV-66.02".FB_OPEN OR "IO_Valve_Buffer_DB"."AV-66.03".FB_OPEN);
   "BFT-66".IN_FBAV_CIP_Tank := "AlwaysTRUE" AND "IO_Valve_Buffer_DB"."AV-65.21".FB_OPEN AND ("IO_Valve_Buffer_DB"."AV-66.04".FB_OPEN OR "IO_Valve_Buffer_DB"."AV-66.05".FB_OPEN);
   "BFT-66".IN_FBAV_CIP_Line := "AlwaysTRUE" AND "IO_Valve_Buffer_DB"."AV-65.21".FB_OPEN;
END_REGION

REGION Network 15: Comm BFT 65 and BFT 66 to Blending
   RUNG wire#powerrail
      Contact( "AlwaysTRUE" )
      wire#w1
      Contact( "BFT-65".Out_Prod_Req )
      wire#w2
      Coil( "Blend_T-31"."BFT-2 Prod Req" )
   END_RUNG
   RUNG wire#w1
      Contact( "BFT-66".Out_Prod_Req )
   END_RUNG wire#w2
   RUNG wire#w2
      Coil( "Blend_T-40"."BFT-2 Prod Req" )
   END_RUNG
   RUNG wire#w2
      Coil( "Blend_T-41"."BFT-2 Prod Req" )
   END_RUNG
   RUNG wire#w1
      Contact( "BFT-65".Out_Prod_LineOpen )
      wire#w3
      Coil( "Blend_T-31"."BFT-2 Prod Line" )
   END_RUNG
   RUNG wire#w1
      Contact( "BFT-66".Out_Prod_LineOpen )
   END_RUNG wire#w3
   RUNG wire#w3
      Coil( "Blend_T-40"."BFT-2 Prod Line" )
   END_RUNG
   RUNG wire#w3
      Coil( "Blend_T-41"."BFT-2 Prod Line" )
   END_RUNG
   // the same network as SCL:
   "Blend_T-31"."BFT-2 Prod Req" := "AlwaysTRUE" AND ("BFT-65".Out_Prod_Req OR "BFT-66".Out_Prod_Req);
   "Blend_T-40"."BFT-2 Prod Req" := "Blend_T-31"."BFT-2 Prod Req";
   "Blend_T-41"."BFT-2 Prod Req" := "Blend_T-31"."BFT-2 Prod Req";
   "Blend_T-31"."BFT-2 Prod Line" := "AlwaysTRUE" AND ("BFT-65".Out_Prod_LineOpen OR "BFT-66".Out_Prod_LineOpen);
   "Blend_T-40"."BFT-2 Prod Line" := "Blend_T-31"."BFT-2 Prod Line";
   "Blend_T-41"."BFT-2 Prod Line" := "Blend_T-31"."BFT-2 Prod Line";
END_REGION

REGION Network 16: Comm CIP Line 65 & 66
   RUNG wire#powerrail
      Contact( "AlwaysTRUE" )
      wire#w1
      Contact( "BFT-65".Out_CIP_Line_Req )
      wire#w2
      Coil( "Mix_to_CIP".CIP_Request."Buffer Cluster 2"."T65&T66_CIP_LineToPasteur_Request" )
   END_RUNG
   RUNG wire#w1
      Contact( "BFT-66".Out_CIP_Line_Req )
   END_RUNG wire#w2
   RUNG wire#w1
      Contact( "BFT-65".Out_CIP_Line_LineOpen )
      wire#w3
      Coil( "Mix_to_CIP".CIP_Line_OK."Buffer Cluster 2"."T65&T66_CIP_LineToPasteur_LineOK" )
   END_RUNG
   RUNG wire#w1
      Contact( "BFT-66".Out_CIP_Line_LineOpen )
   END_RUNG wire#w3
   // the same network as SCL:
   "Mix_to_CIP".CIP_Request."Buffer Cluster 2"."T65&T66_CIP_LineToPasteur_Request" := "AlwaysTRUE" AND ("BFT-65".Out_CIP_Line_Req OR "BFT-66".Out_CIP_Line_Req);
   "Mix_to_CIP".CIP_Line_OK."Buffer Cluster 2"."T65&T66_CIP_LineToPasteur_LineOK" := "AlwaysTRUE" AND ("BFT-65".Out_CIP_Line_LineOpen OR "BFT-66".Out_CIP_Line_LineOpen);
END_REGION

REGION Network 18: BFT 67
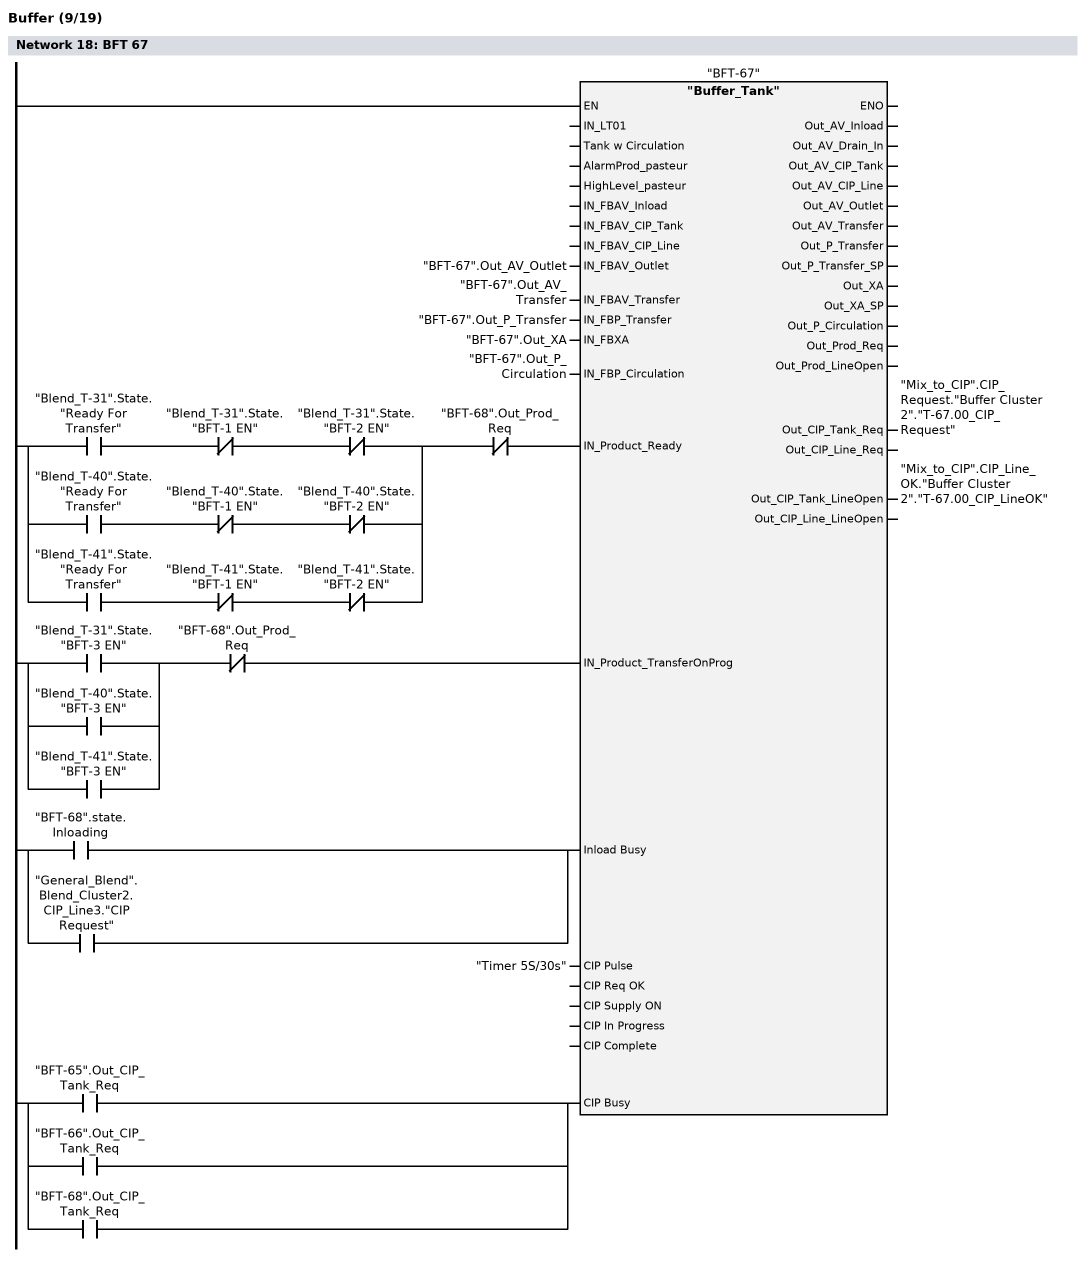
   RUNG wire#powerrail
      "BFT-67"(IN_Product_Ready := wire#w2, IN_Product_TransferOnProg := wire#w4, "Inload Busy" := wire#w5, "CIP Busy" := wire#w6, IN_LT01 :=, "Tank w Circulation" :=, AlarmProd_pasteur :=, HighLevel_pasteur :=, IN_FBAV_Inload :=, IN_FBAV_CIP_Tank :=, IN_FBAV_CIP_Line :=, IN_FBAV_Outlet := "BFT-67".Out_AV_Outlet, IN_FBAV_Transfer := "BFT-67".Out_AV_Transfer, IN_FBP_Transfer := "BFT-67".Out_P_Transfer, IN_FBXA := "BFT-67".Out_XA, IN_FBP_Circulation := "BFT-67".Out_P_Circulation, "CIP Pulse" := "Timer 5S/30s", "CIP Req OK" :=, "CIP Supply ON" :=, "CIP In Progress" :=, "CIP Complete" :=, Out_AV_Inload =>, Out_AV_Drain_In =>, Out_AV_CIP_Tank =>, Out_AV_CIP_Line =>, Out_AV_Outlet =>, Out_AV_Transfer =>, Out_P_Transfer =>, Out_P_Transfer_SP =>, Out_XA =>, Out_XA_SP =>, Out_P_Circulation =>, Out_Prod_Req =>, Out_Prod_LineOpen =>, Out_CIP_Tank_Req => "Mix_to_CIP".CIP_Request."Buffer Cluster 2"."T-67.00_CIP_Request", Out_CIP_Line_Req =>, Out_CIP_Tank_LineOpen => "Mix_to_CIP".CIP_Line_OK."Buffer Cluster 2"."T-67.00_CIP_LineOK", Out_CIP_Line_LineOpen =>)
   END_RUNG
   RUNG wire#powerrail
      Contact( "Blend_T-31".State."Ready For Transfer" )
      I_Contact( "Blend_T-31".State."BFT-1 EN" )
      I_Contact( "Blend_T-31".State."BFT-2 EN" )
      wire#w1
      I_Contact( "BFT-68".Out_Prod_Req )
   END_RUNG wire#w2
   RUNG wire#powerrail
      Contact( "Blend_T-40".State."Ready For Transfer" )
      I_Contact( "Blend_T-40".State."BFT-1 EN" )
      I_Contact( "Blend_T-40".State."BFT-2 EN" )
   END_RUNG wire#w1
   RUNG wire#powerrail
      Contact( "Blend_T-41".State."Ready For Transfer" )
      I_Contact( "Blend_T-41".State."BFT-1 EN" )
      I_Contact( "Blend_T-41".State."BFT-2 EN" )
   END_RUNG wire#w1
   RUNG wire#powerrail
      Contact( "Blend_T-31".State."BFT-3 EN" )
      wire#w3
      I_Contact( "BFT-68".Out_Prod_Req )
   END_RUNG wire#w4
   RUNG wire#powerrail
      Contact( "Blend_T-40".State."BFT-3 EN" )
   END_RUNG wire#w3
   RUNG wire#powerrail
      Contact( "Blend_T-41".State."BFT-3 EN" )
   END_RUNG wire#w3
   RUNG wire#powerrail
      Contact( "BFT-68".state.Inloading )
   END_RUNG wire#w5
   RUNG wire#powerrail
      Contact( "General_Blend".Blend_Cluster2.CIP_Line3."CIP Request" )
   END_RUNG wire#w5
   RUNG wire#powerrail
      Contact( "BFT-65".Out_CIP_Tank_Req )
   END_RUNG wire#w6
   RUNG wire#powerrail
      Contact( "BFT-66".Out_CIP_Tank_Req )
   END_RUNG wire#w6
   RUNG wire#powerrail
      Contact( "BFT-68".Out_CIP_Tank_Req )
   END_RUNG wire#w6
   // the same network as SCL:
   "BFT-67"(IN_FBAV_Outlet := "BFT-67".Out_AV_Outlet,   // "Buffer_Tank"
            IN_FBAV_Transfer := "BFT-67".Out_AV_Transfer,
            IN_FBP_Transfer := "BFT-67".Out_P_Transfer,
            IN_FBXA := "BFT-67".Out_XA,
            IN_FBP_Circulation := "BFT-67".Out_P_Circulation,
            IN_Product_Ready := (("Blend_T-31".State."Ready For Transfer" AND NOT "Blend_T-31".State."BFT-1 EN" AND NOT "Blend_T-31".State."BFT-2 EN") OR ("Blend_T-40".State."Ready For Transfer" AND NOT "Blend_T-40".State."BFT-1 EN" AND NOT "Blend_T-40".State."BFT-2 EN") OR ("Blend_T-41".State."Ready For Transfer" AND NOT "Blend_T-41".State."BFT-1 EN" AND NOT "Blend_T-41".State."BFT-2 EN")) AND NOT "BFT-68".Out_Prod_Req,
            IN_Product_TransferOnProg := ("Blend_T-31".State."BFT-3 EN" OR "Blend_T-40".State."BFT-3 EN" OR "Blend_T-41".State."BFT-3 EN") AND NOT "BFT-68".Out_Prod_Req,
            "Inload Busy" := "BFT-68".state.Inloading OR "General_Blend".Blend_Cluster2.CIP_Line3."CIP Request",
            "CIP Pulse" := "Timer 5S/30s",
            "CIP Busy" := "BFT-65".Out_CIP_Tank_Req OR "BFT-66".Out_CIP_Tank_Req OR "BFT-68".Out_CIP_Tank_Req,
            Out_CIP_Tank_Req => "Mix_to_CIP".CIP_Request."Buffer Cluster 2"."T-67.00_CIP_Request",
            Out_CIP_Tank_LineOpen => "Mix_to_CIP".CIP_Line_OK."Buffer Cluster 2"."T-67.00_CIP_LineOK");
END_REGION

REGION Network 19: BFT 67 Feedback Instrument
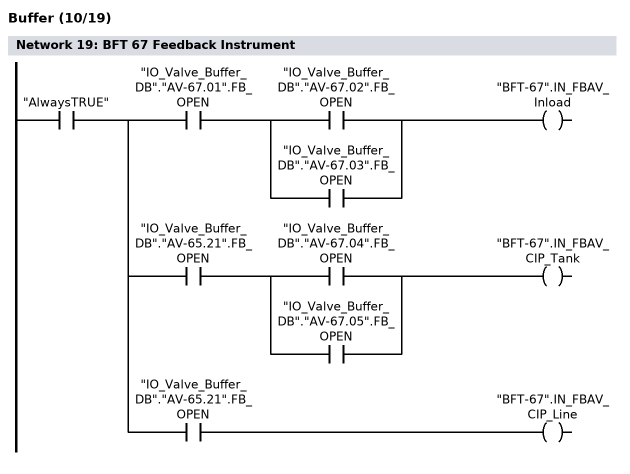
   RUNG wire#powerrail
      Contact( "AlwaysTRUE" )
      wire#w1
      Contact( "IO_Valve_Buffer_DB"."AV-67.01".FB_OPEN )
      wire#w2
      Contact( "IO_Valve_Buffer_DB"."AV-67.02".FB_OPEN )
      wire#w3
      Coil( "BFT-67".IN_FBAV_Inload )
   END_RUNG
   RUNG wire#w2
      Contact( "IO_Valve_Buffer_DB"."AV-67.03".FB_OPEN )
   END_RUNG wire#w3
   RUNG wire#w1
      Contact( "IO_Valve_Buffer_DB"."AV-65.21".FB_OPEN )
      wire#w4
      Contact( "IO_Valve_Buffer_DB"."AV-67.04".FB_OPEN )
      wire#w5
      Coil( "BFT-67".IN_FBAV_CIP_Tank )
   END_RUNG
   RUNG wire#w4
      Contact( "IO_Valve_Buffer_DB"."AV-67.05".FB_OPEN )
   END_RUNG wire#w5
   RUNG wire#w1
      Contact( "IO_Valve_Buffer_DB"."AV-65.21".FB_OPEN )
      Coil( "BFT-67".IN_FBAV_CIP_Line )
   END_RUNG
   // the same network as SCL:
   "BFT-67".IN_FBAV_Inload := "AlwaysTRUE" AND "IO_Valve_Buffer_DB"."AV-67.01".FB_OPEN AND ("IO_Valve_Buffer_DB"."AV-67.02".FB_OPEN OR "IO_Valve_Buffer_DB"."AV-67.03".FB_OPEN);
   "BFT-67".IN_FBAV_CIP_Tank := "AlwaysTRUE" AND "IO_Valve_Buffer_DB"."AV-65.21".FB_OPEN AND ("IO_Valve_Buffer_DB"."AV-67.04".FB_OPEN OR "IO_Valve_Buffer_DB"."AV-67.05".FB_OPEN);
   "BFT-67".IN_FBAV_CIP_Line := "AlwaysTRUE" AND "IO_Valve_Buffer_DB"."AV-65.21".FB_OPEN;
END_REGION

REGION Network 20: BFT 68
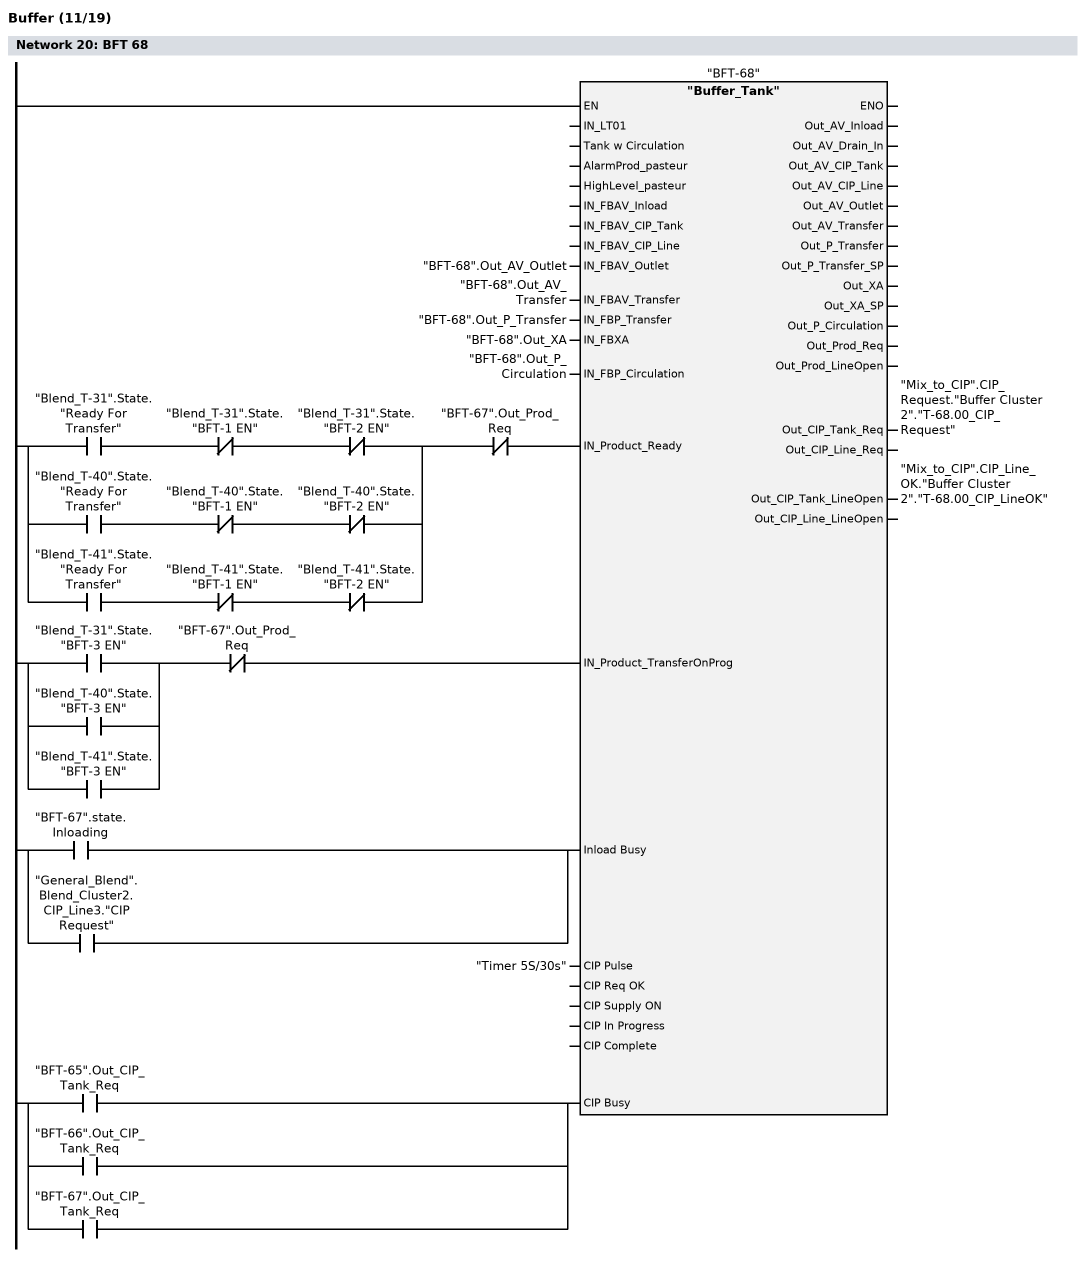
   RUNG wire#powerrail
      "BFT-68"(IN_Product_Ready := wire#w2, IN_Product_TransferOnProg := wire#w4, "Inload Busy" := wire#w5, "CIP Busy" := wire#w6, IN_LT01 :=, "Tank w Circulation" :=, AlarmProd_pasteur :=, HighLevel_pasteur :=, IN_FBAV_Inload :=, IN_FBAV_CIP_Tank :=, IN_FBAV_CIP_Line :=, IN_FBAV_Outlet := "BFT-68".Out_AV_Outlet, IN_FBAV_Transfer := "BFT-68".Out_AV_Transfer, IN_FBP_Transfer := "BFT-68".Out_P_Transfer, IN_FBXA := "BFT-68".Out_XA, IN_FBP_Circulation := "BFT-68".Out_P_Circulation, "CIP Pulse" := "Timer 5S/30s", "CIP Req OK" :=, "CIP Supply ON" :=, "CIP In Progress" :=, "CIP Complete" :=, Out_AV_Inload =>, Out_AV_Drain_In =>, Out_AV_CIP_Tank =>, Out_AV_CIP_Line =>, Out_AV_Outlet =>, Out_AV_Transfer =>, Out_P_Transfer =>, Out_P_Transfer_SP =>, Out_XA =>, Out_XA_SP =>, Out_P_Circulation =>, Out_Prod_Req =>, Out_Prod_LineOpen =>, Out_CIP_Tank_Req => "Mix_to_CIP".CIP_Request."Buffer Cluster 2"."T-68.00_CIP_Request", Out_CIP_Line_Req =>, Out_CIP_Tank_LineOpen => "Mix_to_CIP".CIP_Line_OK."Buffer Cluster 2"."T-68.00_CIP_LineOK", Out_CIP_Line_LineOpen =>)
   END_RUNG
   RUNG wire#powerrail
      Contact( "Blend_T-31".State."Ready For Transfer" )
      I_Contact( "Blend_T-31".State."BFT-1 EN" )
      I_Contact( "Blend_T-31".State."BFT-2 EN" )
      wire#w1
      I_Contact( "BFT-67".Out_Prod_Req )
   END_RUNG wire#w2
   RUNG wire#powerrail
      Contact( "Blend_T-40".State."Ready For Transfer" )
      I_Contact( "Blend_T-40".State."BFT-1 EN" )
      I_Contact( "Blend_T-40".State."BFT-2 EN" )
   END_RUNG wire#w1
   RUNG wire#powerrail
      Contact( "Blend_T-41".State."Ready For Transfer" )
      I_Contact( "Blend_T-41".State."BFT-1 EN" )
      I_Contact( "Blend_T-41".State."BFT-2 EN" )
   END_RUNG wire#w1
   RUNG wire#powerrail
      Contact( "Blend_T-31".State."BFT-3 EN" )
      wire#w3
      I_Contact( "BFT-67".Out_Prod_Req )
   END_RUNG wire#w4
   RUNG wire#powerrail
      Contact( "Blend_T-40".State."BFT-3 EN" )
   END_RUNG wire#w3
   RUNG wire#powerrail
      Contact( "Blend_T-41".State."BFT-3 EN" )
   END_RUNG wire#w3
   RUNG wire#powerrail
      Contact( "BFT-67".state.Inloading )
   END_RUNG wire#w5
   RUNG wire#powerrail
      Contact( "General_Blend".Blend_Cluster2.CIP_Line3."CIP Request" )
   END_RUNG wire#w5
   RUNG wire#powerrail
      Contact( "BFT-65".Out_CIP_Tank_Req )
   END_RUNG wire#w6
   RUNG wire#powerrail
      Contact( "BFT-66".Out_CIP_Tank_Req )
   END_RUNG wire#w6
   RUNG wire#powerrail
      Contact( "BFT-67".Out_CIP_Tank_Req )
   END_RUNG wire#w6
   // the same network as SCL:
   "BFT-68"(IN_FBAV_Outlet := "BFT-68".Out_AV_Outlet,   // "Buffer_Tank"
            IN_FBAV_Transfer := "BFT-68".Out_AV_Transfer,
            IN_FBP_Transfer := "BFT-68".Out_P_Transfer,
            IN_FBXA := "BFT-68".Out_XA,
            IN_FBP_Circulation := "BFT-68".Out_P_Circulation,
            IN_Product_Ready := (("Blend_T-31".State."Ready For Transfer" AND NOT "Blend_T-31".State."BFT-1 EN" AND NOT "Blend_T-31".State."BFT-2 EN") OR ("Blend_T-40".State."Ready For Transfer" AND NOT "Blend_T-40".State."BFT-1 EN" AND NOT "Blend_T-40".State."BFT-2 EN") OR ("Blend_T-41".State."Ready For Transfer" AND NOT "Blend_T-41".State."BFT-1 EN" AND NOT "Blend_T-41".State."BFT-2 EN")) AND NOT "BFT-67".Out_Prod_Req,
            IN_Product_TransferOnProg := ("Blend_T-31".State."BFT-3 EN" OR "Blend_T-40".State."BFT-3 EN" OR "Blend_T-41".State."BFT-3 EN") AND NOT "BFT-67".Out_Prod_Req,
            "Inload Busy" := "BFT-67".state.Inloading OR "General_Blend".Blend_Cluster2.CIP_Line3."CIP Request",
            "CIP Pulse" := "Timer 5S/30s",
            "CIP Busy" := "BFT-65".Out_CIP_Tank_Req OR "BFT-66".Out_CIP_Tank_Req OR "BFT-67".Out_CIP_Tank_Req,
            Out_CIP_Tank_Req => "Mix_to_CIP".CIP_Request."Buffer Cluster 2"."T-68.00_CIP_Request",
            Out_CIP_Tank_LineOpen => "Mix_to_CIP".CIP_Line_OK."Buffer Cluster 2"."T-68.00_CIP_LineOK");
END_REGION

REGION Network 21: BFT 68 Feedback Instrument
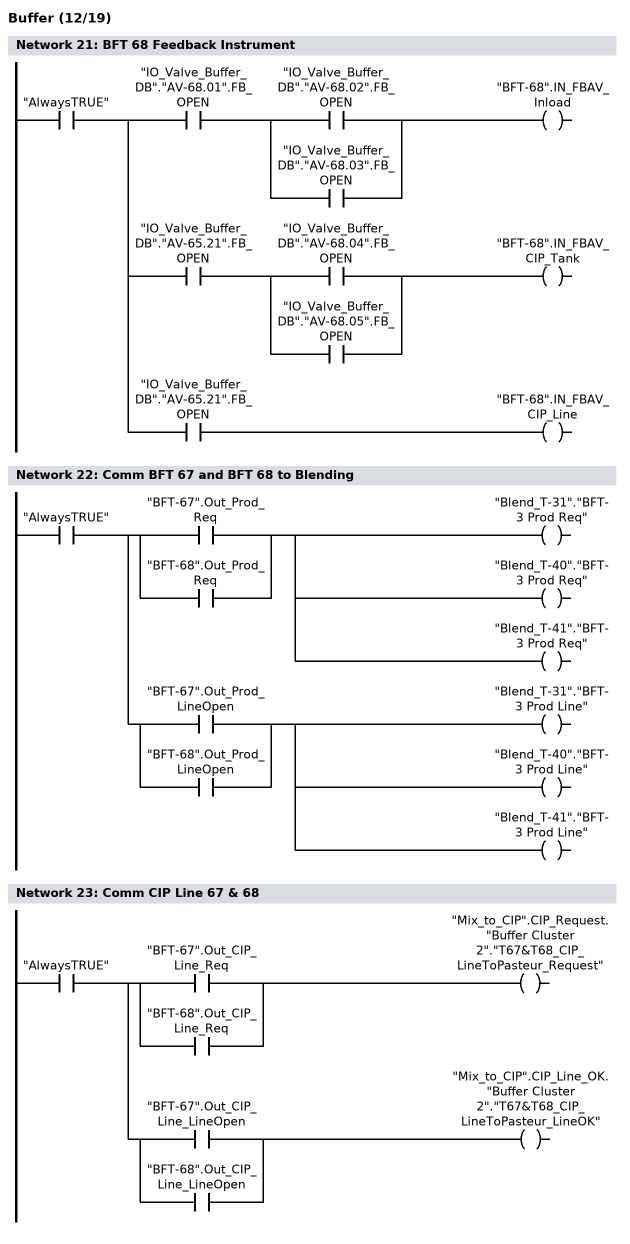
   RUNG wire#powerrail
      Contact( "AlwaysTRUE" )
      wire#w1
      Contact( "IO_Valve_Buffer_DB"."AV-68.01".FB_OPEN )
      wire#w2
      Contact( "IO_Valve_Buffer_DB"."AV-68.02".FB_OPEN )
      wire#w3
      Coil( "BFT-68".IN_FBAV_Inload )
   END_RUNG
   RUNG wire#w2
      Contact( "IO_Valve_Buffer_DB"."AV-68.03".FB_OPEN )
   END_RUNG wire#w3
   RUNG wire#w1
      Contact( "IO_Valve_Buffer_DB"."AV-65.21".FB_OPEN )
      wire#w4
      Contact( "IO_Valve_Buffer_DB"."AV-68.04".FB_OPEN )
      wire#w5
      Coil( "BFT-68".IN_FBAV_CIP_Tank )
   END_RUNG
   RUNG wire#w4
      Contact( "IO_Valve_Buffer_DB"."AV-68.05".FB_OPEN )
   END_RUNG wire#w5
   RUNG wire#w1
      Contact( "IO_Valve_Buffer_DB"."AV-65.21".FB_OPEN )
      Coil( "BFT-68".IN_FBAV_CIP_Line )
   END_RUNG
   // the same network as SCL:
   "BFT-68".IN_FBAV_Inload := "AlwaysTRUE" AND "IO_Valve_Buffer_DB"."AV-68.01".FB_OPEN AND ("IO_Valve_Buffer_DB"."AV-68.02".FB_OPEN OR "IO_Valve_Buffer_DB"."AV-68.03".FB_OPEN);
   "BFT-68".IN_FBAV_CIP_Tank := "AlwaysTRUE" AND "IO_Valve_Buffer_DB"."AV-65.21".FB_OPEN AND ("IO_Valve_Buffer_DB"."AV-68.04".FB_OPEN OR "IO_Valve_Buffer_DB"."AV-68.05".FB_OPEN);
   "BFT-68".IN_FBAV_CIP_Line := "AlwaysTRUE" AND "IO_Valve_Buffer_DB"."AV-65.21".FB_OPEN;
END_REGION

REGION Network 22: Comm BFT 67 and BFT 68 to Blending
   RUNG wire#powerrail
      Contact( "AlwaysTRUE" )
      wire#w1
      Contact( "BFT-67".Out_Prod_Req )
      wire#w2
      Coil( "Blend_T-31"."BFT-3 Prod Req" )
   END_RUNG
   RUNG wire#w1
      Contact( "BFT-68".Out_Prod_Req )
   END_RUNG wire#w2
   RUNG wire#w2
      Coil( "Blend_T-40"."BFT-3 Prod Req" )
   END_RUNG
   RUNG wire#w2
      Coil( "Blend_T-41"."BFT-3 Prod Req" )
   END_RUNG
   RUNG wire#w1
      Contact( "BFT-67".Out_Prod_LineOpen )
      wire#w3
      Coil( "Blend_T-31"."BFT-3 Prod Line" )
   END_RUNG
   RUNG wire#w1
      Contact( "BFT-68".Out_Prod_LineOpen )
   END_RUNG wire#w3
   RUNG wire#w3
      Coil( "Blend_T-40"."BFT-3 Prod Line" )
   END_RUNG
   RUNG wire#w3
      Coil( "Blend_T-41"."BFT-3 Prod Line" )
   END_RUNG
   // the same network as SCL:
   "Blend_T-31"."BFT-3 Prod Req" := "AlwaysTRUE" AND ("BFT-67".Out_Prod_Req OR "BFT-68".Out_Prod_Req);
   "Blend_T-40"."BFT-3 Prod Req" := "Blend_T-31"."BFT-3 Prod Req";
   "Blend_T-41"."BFT-3 Prod Req" := "Blend_T-31"."BFT-3 Prod Req";
   "Blend_T-31"."BFT-3 Prod Line" := "AlwaysTRUE" AND ("BFT-67".Out_Prod_LineOpen OR "BFT-68".Out_Prod_LineOpen);
   "Blend_T-40"."BFT-3 Prod Line" := "Blend_T-31"."BFT-3 Prod Line";
   "Blend_T-41"."BFT-3 Prod Line" := "Blend_T-31"."BFT-3 Prod Line";
END_REGION

REGION Network 23: Comm CIP Line 67 & 68
   RUNG wire#powerrail
      Contact( "AlwaysTRUE" )
      wire#w1
      Contact( "BFT-67".Out_CIP_Line_Req )
      wire#w2
      Coil( "Mix_to_CIP".CIP_Request."Buffer Cluster 2"."T67&T68_CIP_LineToPasteur_Request" )
   END_RUNG
   RUNG wire#w1
      Contact( "BFT-68".Out_CIP_Line_Req )
   END_RUNG wire#w2
   RUNG wire#w1
      Contact( "BFT-67".Out_CIP_Line_LineOpen )
      wire#w3
      Coil( "Mix_to_CIP".CIP_Line_OK."Buffer Cluster 2"."T67&T68_CIP_LineToPasteur_LineOK" )
   END_RUNG
   RUNG wire#w1
      Contact( "BFT-68".Out_CIP_Line_LineOpen )
   END_RUNG wire#w3
   // the same network as SCL:
   "Mix_to_CIP".CIP_Request."Buffer Cluster 2"."T67&T68_CIP_LineToPasteur_Request" := "AlwaysTRUE" AND ("BFT-67".Out_CIP_Line_Req OR "BFT-68".Out_CIP_Line_Req);
   "Mix_to_CIP".CIP_Line_OK."Buffer Cluster 2"."T67&T68_CIP_LineToPasteur_LineOK" := "AlwaysTRUE" AND ("BFT-67".Out_CIP_Line_LineOpen OR "BFT-68".Out_CIP_Line_LineOpen);
END_REGION

REGION Network 25: Comm CIP to BFT 61 Rework 32
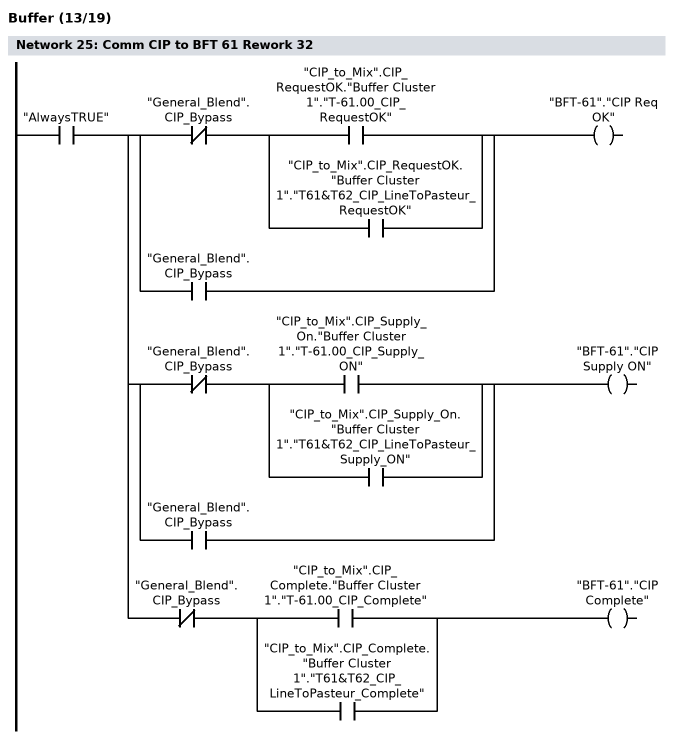
   RUNG wire#powerrail
      Contact( "AlwaysTRUE" )
      wire#w1
      I_Contact( "General_Blend".CIP_Bypass )
      wire#w2
      Contact( "CIP_to_Mix".CIP_RequestOK."Buffer Cluster 1"."T-61.00_CIP_RequestOK" )
      wire#w3
      Coil( "BFT-61"."CIP Req OK" )
   END_RUNG
   RUNG wire#w2
      Contact( "CIP_to_Mix".CIP_RequestOK."Buffer Cluster 1"."T61&T62_CIP_LineToPasteur_RequestOK" )
   END_RUNG wire#w3
   RUNG wire#w1
      Contact( "General_Blend".CIP_Bypass )
   END_RUNG wire#w3
   RUNG wire#w1
      I_Contact( "General_Blend".CIP_Bypass )
      wire#w4
      Contact( "CIP_to_Mix".CIP_Supply_On."Buffer Cluster 1"."T-61.00_CIP_Supply_ON" )
      wire#w5
      Coil( "BFT-61"."CIP Supply ON" )
   END_RUNG
   RUNG wire#w4
      Contact( "CIP_to_Mix".CIP_Supply_On."Buffer Cluster 1"."T61&T62_CIP_LineToPasteur_Supply_ON" )
   END_RUNG wire#w5
   RUNG wire#w1
      Contact( "General_Blend".CIP_Bypass )
   END_RUNG wire#w5
   RUNG wire#w1
      I_Contact( "General_Blend".CIP_Bypass )
      wire#w6
      Contact( "CIP_to_Mix".CIP_Complete."Buffer Cluster 1"."T-61.00_CIP_Complete" )
      wire#w7
      Coil( "BFT-61"."CIP Complete" )
   END_RUNG
   RUNG wire#w6
      Contact( "CIP_to_Mix".CIP_Complete."Buffer Cluster 1"."T61&T62_CIP_LineToPasteur_Complete" )
   END_RUNG wire#w7
   // the same network as SCL:
   "BFT-61"."CIP Req OK" := "AlwaysTRUE" AND ((NOT "General_Blend".CIP_Bypass AND ("CIP_to_Mix".CIP_RequestOK."Buffer Cluster 1"."T-61.00_CIP_RequestOK" OR "CIP_to_Mix".CIP_RequestOK."Buffer Cluster 1"."T61&T62_CIP_LineToPasteur_RequestOK")) OR "General_Blend".CIP_Bypass);
   "BFT-61"."CIP Supply ON" := "AlwaysTRUE" AND ((NOT "General_Blend".CIP_Bypass AND ("CIP_to_Mix".CIP_Supply_On."Buffer Cluster 1"."T-61.00_CIP_Supply_ON" OR "CIP_to_Mix".CIP_Supply_On."Buffer Cluster 1"."T61&T62_CIP_LineToPasteur_Supply_ON")) OR "General_Blend".CIP_Bypass);
   "BFT-61"."CIP Complete" := "AlwaysTRUE" AND NOT "General_Blend".CIP_Bypass AND ("CIP_to_Mix".CIP_Complete."Buffer Cluster 1"."T-61.00_CIP_Complete" OR "CIP_to_Mix".CIP_Complete."Buffer Cluster 1"."T61&T62_CIP_LineToPasteur_Complete");
END_REGION

REGION Network 26: Comm CIP to BFT 64 Rework 22
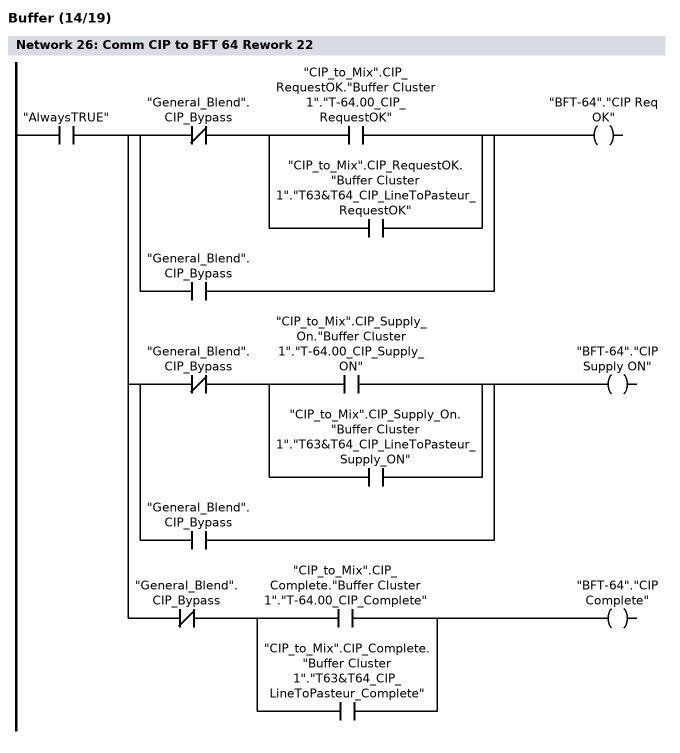
   RUNG wire#powerrail
      Contact( "AlwaysTRUE" )
      wire#w1
      I_Contact( "General_Blend".CIP_Bypass )
      wire#w2
      Contact( "CIP_to_Mix".CIP_RequestOK."Buffer Cluster 1"."T-64.00_CIP_RequestOK" )
      wire#w3
      Coil( "BFT-64"."CIP Req OK" )
   END_RUNG
   RUNG wire#w2
      Contact( "CIP_to_Mix".CIP_RequestOK."Buffer Cluster 1"."T63&T64_CIP_LineToPasteur_RequestOK" )
   END_RUNG wire#w3
   RUNG wire#w1
      Contact( "General_Blend".CIP_Bypass )
   END_RUNG wire#w3
   RUNG wire#w1
      I_Contact( "General_Blend".CIP_Bypass )
      wire#w4
      Contact( "CIP_to_Mix".CIP_Supply_On."Buffer Cluster 1"."T-64.00_CIP_Supply_ON" )
      wire#w5
      Coil( "BFT-64"."CIP Supply ON" )
   END_RUNG
   RUNG wire#w4
      Contact( "CIP_to_Mix".CIP_Supply_On."Buffer Cluster 1"."T63&T64_CIP_LineToPasteur_Supply_ON" )
   END_RUNG wire#w5
   RUNG wire#w1
      Contact( "General_Blend".CIP_Bypass )
   END_RUNG wire#w5
   RUNG wire#w1
      I_Contact( "General_Blend".CIP_Bypass )
      wire#w6
      Contact( "CIP_to_Mix".CIP_Complete."Buffer Cluster 1"."T-64.00_CIP_Complete" )
      wire#w7
      Coil( "BFT-64"."CIP Complete" )
   END_RUNG
   RUNG wire#w6
      Contact( "CIP_to_Mix".CIP_Complete."Buffer Cluster 1"."T63&T64_CIP_LineToPasteur_Complete" )
   END_RUNG wire#w7
   // the same network as SCL:
   "BFT-64"."CIP Req OK" := "AlwaysTRUE" AND ((NOT "General_Blend".CIP_Bypass AND ("CIP_to_Mix".CIP_RequestOK."Buffer Cluster 1"."T-64.00_CIP_RequestOK" OR "CIP_to_Mix".CIP_RequestOK."Buffer Cluster 1"."T63&T64_CIP_LineToPasteur_RequestOK")) OR "General_Blend".CIP_Bypass);
   "BFT-64"."CIP Supply ON" := "AlwaysTRUE" AND ((NOT "General_Blend".CIP_Bypass AND ("CIP_to_Mix".CIP_Supply_On."Buffer Cluster 1"."T-64.00_CIP_Supply_ON" OR "CIP_to_Mix".CIP_Supply_On."Buffer Cluster 1"."T63&T64_CIP_LineToPasteur_Supply_ON")) OR "General_Blend".CIP_Bypass);
   "BFT-64"."CIP Complete" := "AlwaysTRUE" AND NOT "General_Blend".CIP_Bypass AND ("CIP_to_Mix".CIP_Complete."Buffer Cluster 1"."T-64.00_CIP_Complete" OR "CIP_to_Mix".CIP_Complete."Buffer Cluster 1"."T63&T64_CIP_LineToPasteur_Complete");
END_REGION

REGION Network 27: Comm CIP to BFT 65
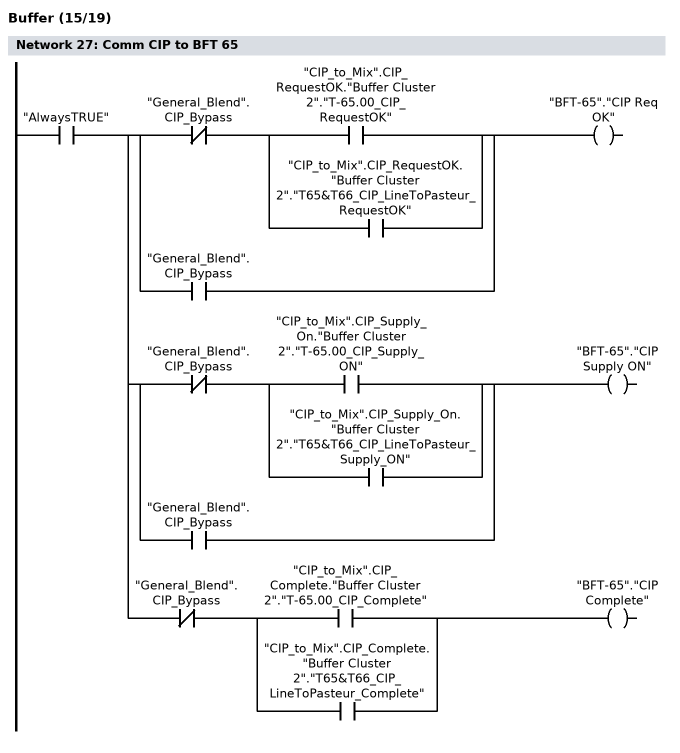
   RUNG wire#powerrail
      Contact( "AlwaysTRUE" )
      wire#w1
      I_Contact( "General_Blend".CIP_Bypass )
      wire#w2
      Contact( "CIP_to_Mix".CIP_RequestOK."Buffer Cluster 2"."T-65.00_CIP_RequestOK" )
      wire#w3
      Coil( "BFT-65"."CIP Req OK" )
   END_RUNG
   RUNG wire#w2
      Contact( "CIP_to_Mix".CIP_RequestOK."Buffer Cluster 2"."T65&T66_CIP_LineToPasteur_RequestOK" )
   END_RUNG wire#w3
   RUNG wire#w1
      Contact( "General_Blend".CIP_Bypass )
   END_RUNG wire#w3
   RUNG wire#w1
      I_Contact( "General_Blend".CIP_Bypass )
      wire#w4
      Contact( "CIP_to_Mix".CIP_Supply_On."Buffer Cluster 2"."T-65.00_CIP_Supply_ON" )
      wire#w5
      Coil( "BFT-65"."CIP Supply ON" )
   END_RUNG
   RUNG wire#w4
      Contact( "CIP_to_Mix".CIP_Supply_On."Buffer Cluster 2"."T65&T66_CIP_LineToPasteur_Supply_ON" )
   END_RUNG wire#w5
   RUNG wire#w1
      Contact( "General_Blend".CIP_Bypass )
   END_RUNG wire#w5
   RUNG wire#w1
      I_Contact( "General_Blend".CIP_Bypass )
      wire#w6
      Contact( "CIP_to_Mix".CIP_Complete."Buffer Cluster 2"."T-65.00_CIP_Complete" )
      wire#w7
      Coil( "BFT-65"."CIP Complete" )
   END_RUNG
   RUNG wire#w6
      Contact( "CIP_to_Mix".CIP_Complete."Buffer Cluster 2"."T65&T66_CIP_LineToPasteur_Complete" )
   END_RUNG wire#w7
   // the same network as SCL:
   "BFT-65"."CIP Req OK" := "AlwaysTRUE" AND ((NOT "General_Blend".CIP_Bypass AND ("CIP_to_Mix".CIP_RequestOK."Buffer Cluster 2"."T-65.00_CIP_RequestOK" OR "CIP_to_Mix".CIP_RequestOK."Buffer Cluster 2"."T65&T66_CIP_LineToPasteur_RequestOK")) OR "General_Blend".CIP_Bypass);
   "BFT-65"."CIP Supply ON" := "AlwaysTRUE" AND ((NOT "General_Blend".CIP_Bypass AND ("CIP_to_Mix".CIP_Supply_On."Buffer Cluster 2"."T-65.00_CIP_Supply_ON" OR "CIP_to_Mix".CIP_Supply_On."Buffer Cluster 2"."T65&T66_CIP_LineToPasteur_Supply_ON")) OR "General_Blend".CIP_Bypass);
   "BFT-65"."CIP Complete" := "AlwaysTRUE" AND NOT "General_Blend".CIP_Bypass AND ("CIP_to_Mix".CIP_Complete."Buffer Cluster 2"."T-65.00_CIP_Complete" OR "CIP_to_Mix".CIP_Complete."Buffer Cluster 2"."T65&T66_CIP_LineToPasteur_Complete");
END_REGION

REGION Network 28: Comm CIP to BFT 66
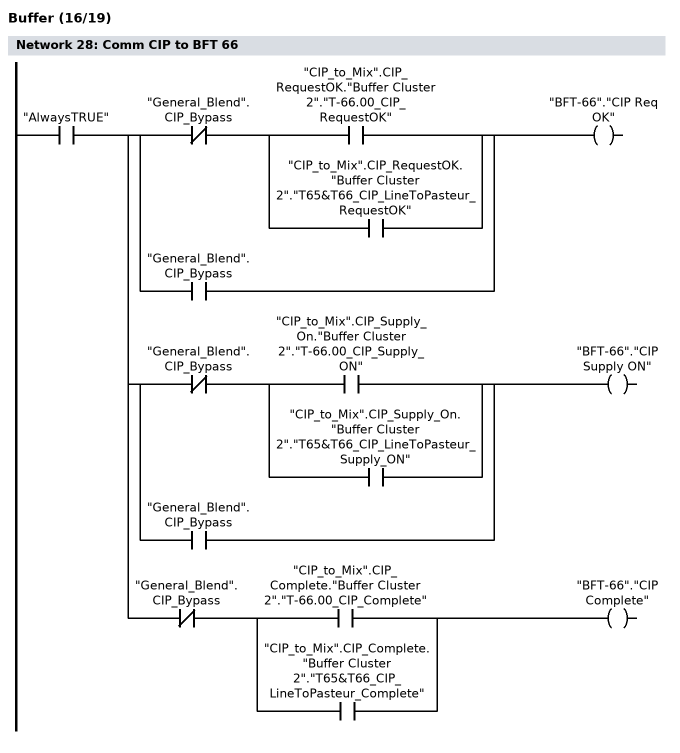
   RUNG wire#powerrail
      Contact( "AlwaysTRUE" )
      wire#w1
      I_Contact( "General_Blend".CIP_Bypass )
      wire#w2
      Contact( "CIP_to_Mix".CIP_RequestOK."Buffer Cluster 2"."T-66.00_CIP_RequestOK" )
      wire#w3
      Coil( "BFT-66"."CIP Req OK" )
   END_RUNG
   RUNG wire#w2
      Contact( "CIP_to_Mix".CIP_RequestOK."Buffer Cluster 2"."T65&T66_CIP_LineToPasteur_RequestOK" )
   END_RUNG wire#w3
   RUNG wire#w1
      Contact( "General_Blend".CIP_Bypass )
   END_RUNG wire#w3
   RUNG wire#w1
      I_Contact( "General_Blend".CIP_Bypass )
      wire#w4
      Contact( "CIP_to_Mix".CIP_Supply_On."Buffer Cluster 2"."T-66.00_CIP_Supply_ON" )
      wire#w5
      Coil( "BFT-66"."CIP Supply ON" )
   END_RUNG
   RUNG wire#w4
      Contact( "CIP_to_Mix".CIP_Supply_On."Buffer Cluster 2"."T65&T66_CIP_LineToPasteur_Supply_ON" )
   END_RUNG wire#w5
   RUNG wire#w1
      Contact( "General_Blend".CIP_Bypass )
   END_RUNG wire#w5
   RUNG wire#w1
      I_Contact( "General_Blend".CIP_Bypass )
      wire#w6
      Contact( "CIP_to_Mix".CIP_Complete."Buffer Cluster 2"."T-66.00_CIP_Complete" )
      wire#w7
      Coil( "BFT-66"."CIP Complete" )
   END_RUNG
   RUNG wire#w6
      Contact( "CIP_to_Mix".CIP_Complete."Buffer Cluster 2"."T65&T66_CIP_LineToPasteur_Complete" )
   END_RUNG wire#w7
   // the same network as SCL:
   "BFT-66"."CIP Req OK" := "AlwaysTRUE" AND ((NOT "General_Blend".CIP_Bypass AND ("CIP_to_Mix".CIP_RequestOK."Buffer Cluster 2"."T-66.00_CIP_RequestOK" OR "CIP_to_Mix".CIP_RequestOK."Buffer Cluster 2"."T65&T66_CIP_LineToPasteur_RequestOK")) OR "General_Blend".CIP_Bypass);
   "BFT-66"."CIP Supply ON" := "AlwaysTRUE" AND ((NOT "General_Blend".CIP_Bypass AND ("CIP_to_Mix".CIP_Supply_On."Buffer Cluster 2"."T-66.00_CIP_Supply_ON" OR "CIP_to_Mix".CIP_Supply_On."Buffer Cluster 2"."T65&T66_CIP_LineToPasteur_Supply_ON")) OR "General_Blend".CIP_Bypass);
   "BFT-66"."CIP Complete" := "AlwaysTRUE" AND NOT "General_Blend".CIP_Bypass AND ("CIP_to_Mix".CIP_Complete."Buffer Cluster 2"."T-66.00_CIP_Complete" OR "CIP_to_Mix".CIP_Complete."Buffer Cluster 2"."T65&T66_CIP_LineToPasteur_Complete");
END_REGION

REGION Network 29: Comm CIP to BFT 67
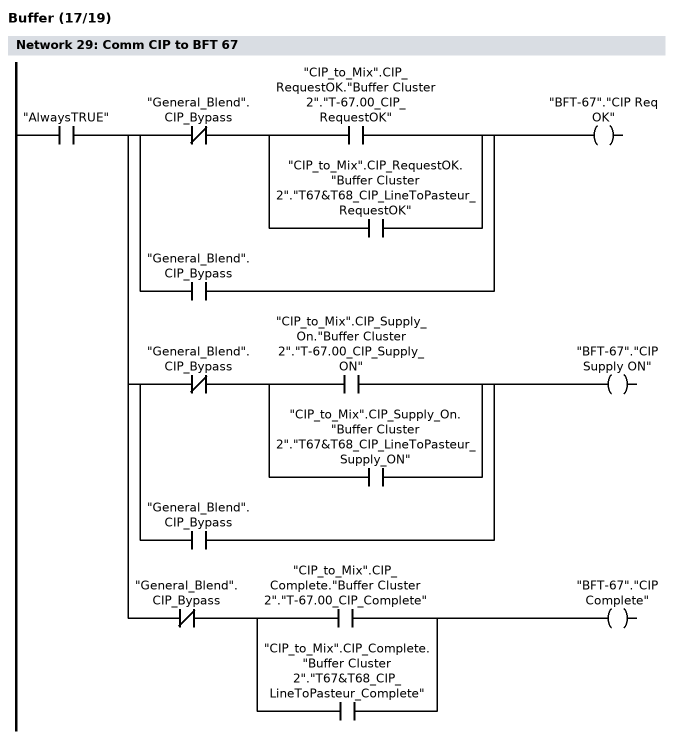
   RUNG wire#powerrail
      Contact( "AlwaysTRUE" )
      wire#w1
      I_Contact( "General_Blend".CIP_Bypass )
      wire#w2
      Contact( "CIP_to_Mix".CIP_RequestOK."Buffer Cluster 2"."T-67.00_CIP_RequestOK" )
      wire#w3
      Coil( "BFT-67"."CIP Req OK" )
   END_RUNG
   RUNG wire#w2
      Contact( "CIP_to_Mix".CIP_RequestOK."Buffer Cluster 2"."T67&T68_CIP_LineToPasteur_RequestOK" )
   END_RUNG wire#w3
   RUNG wire#w1
      Contact( "General_Blend".CIP_Bypass )
   END_RUNG wire#w3
   RUNG wire#w1
      I_Contact( "General_Blend".CIP_Bypass )
      wire#w4
      Contact( "CIP_to_Mix".CIP_Supply_On."Buffer Cluster 2"."T-67.00_CIP_Supply_ON" )
      wire#w5
      Coil( "BFT-67"."CIP Supply ON" )
   END_RUNG
   RUNG wire#w4
      Contact( "CIP_to_Mix".CIP_Supply_On."Buffer Cluster 2"."T67&T68_CIP_LineToPasteur_Supply_ON" )
   END_RUNG wire#w5
   RUNG wire#w1
      Contact( "General_Blend".CIP_Bypass )
   END_RUNG wire#w5
   RUNG wire#w1
      I_Contact( "General_Blend".CIP_Bypass )
      wire#w6
      Contact( "CIP_to_Mix".CIP_Complete."Buffer Cluster 2"."T-67.00_CIP_Complete" )
      wire#w7
      Coil( "BFT-67"."CIP Complete" )
   END_RUNG
   RUNG wire#w6
      Contact( "CIP_to_Mix".CIP_Complete."Buffer Cluster 2"."T67&T68_CIP_LineToPasteur_Complete" )
   END_RUNG wire#w7
   // the same network as SCL:
   "BFT-67"."CIP Req OK" := "AlwaysTRUE" AND ((NOT "General_Blend".CIP_Bypass AND ("CIP_to_Mix".CIP_RequestOK."Buffer Cluster 2"."T-67.00_CIP_RequestOK" OR "CIP_to_Mix".CIP_RequestOK."Buffer Cluster 2"."T67&T68_CIP_LineToPasteur_RequestOK")) OR "General_Blend".CIP_Bypass);
   "BFT-67"."CIP Supply ON" := "AlwaysTRUE" AND ((NOT "General_Blend".CIP_Bypass AND ("CIP_to_Mix".CIP_Supply_On."Buffer Cluster 2"."T-67.00_CIP_Supply_ON" OR "CIP_to_Mix".CIP_Supply_On."Buffer Cluster 2"."T67&T68_CIP_LineToPasteur_Supply_ON")) OR "General_Blend".CIP_Bypass);
   "BFT-67"."CIP Complete" := "AlwaysTRUE" AND NOT "General_Blend".CIP_Bypass AND ("CIP_to_Mix".CIP_Complete."Buffer Cluster 2"."T-67.00_CIP_Complete" OR "CIP_to_Mix".CIP_Complete."Buffer Cluster 2"."T67&T68_CIP_LineToPasteur_Complete");
END_REGION

REGION Network 30: Comm CIP to BFT 68
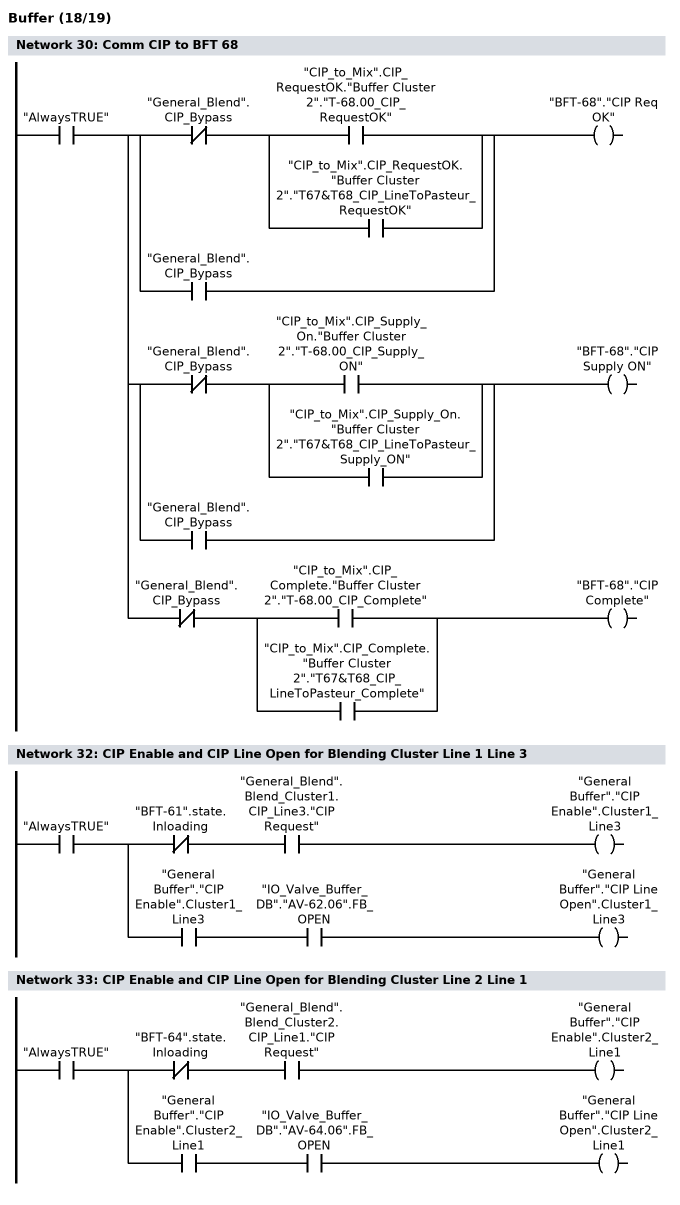
   RUNG wire#powerrail
      Contact( "AlwaysTRUE" )
      wire#w1
      I_Contact( "General_Blend".CIP_Bypass )
      wire#w2
      Contact( "CIP_to_Mix".CIP_RequestOK."Buffer Cluster 2"."T-68.00_CIP_RequestOK" )
      wire#w3
      Coil( "BFT-68"."CIP Req OK" )
   END_RUNG
   RUNG wire#w2
      Contact( "CIP_to_Mix".CIP_RequestOK."Buffer Cluster 2"."T67&T68_CIP_LineToPasteur_RequestOK" )
   END_RUNG wire#w3
   RUNG wire#w1
      Contact( "General_Blend".CIP_Bypass )
   END_RUNG wire#w3
   RUNG wire#w1
      I_Contact( "General_Blend".CIP_Bypass )
      wire#w4
      Contact( "CIP_to_Mix".CIP_Supply_On."Buffer Cluster 2"."T-68.00_CIP_Supply_ON" )
      wire#w5
      Coil( "BFT-68"."CIP Supply ON" )
   END_RUNG
   RUNG wire#w4
      Contact( "CIP_to_Mix".CIP_Supply_On."Buffer Cluster 2"."T67&T68_CIP_LineToPasteur_Supply_ON" )
   END_RUNG wire#w5
   RUNG wire#w1
      Contact( "General_Blend".CIP_Bypass )
   END_RUNG wire#w5
   RUNG wire#w1
      I_Contact( "General_Blend".CIP_Bypass )
      wire#w6
      Contact( "CIP_to_Mix".CIP_Complete."Buffer Cluster 2"."T-68.00_CIP_Complete" )
      wire#w7
      Coil( "BFT-68"."CIP Complete" )
   END_RUNG
   RUNG wire#w6
      Contact( "CIP_to_Mix".CIP_Complete."Buffer Cluster 2"."T67&T68_CIP_LineToPasteur_Complete" )
   END_RUNG wire#w7
   // the same network as SCL:
   "BFT-68"."CIP Req OK" := "AlwaysTRUE" AND ((NOT "General_Blend".CIP_Bypass AND ("CIP_to_Mix".CIP_RequestOK."Buffer Cluster 2"."T-68.00_CIP_RequestOK" OR "CIP_to_Mix".CIP_RequestOK."Buffer Cluster 2"."T67&T68_CIP_LineToPasteur_RequestOK")) OR "General_Blend".CIP_Bypass);
   "BFT-68"."CIP Supply ON" := "AlwaysTRUE" AND ((NOT "General_Blend".CIP_Bypass AND ("CIP_to_Mix".CIP_Supply_On."Buffer Cluster 2"."T-68.00_CIP_Supply_ON" OR "CIP_to_Mix".CIP_Supply_On."Buffer Cluster 2"."T67&T68_CIP_LineToPasteur_Supply_ON")) OR "General_Blend".CIP_Bypass);
   "BFT-68"."CIP Complete" := "AlwaysTRUE" AND NOT "General_Blend".CIP_Bypass AND ("CIP_to_Mix".CIP_Complete."Buffer Cluster 2"."T-68.00_CIP_Complete" OR "CIP_to_Mix".CIP_Complete."Buffer Cluster 2"."T67&T68_CIP_LineToPasteur_Complete");
END_REGION

REGION Network 32: CIP Enable and CIP Line Open for Blending Cluster Line 1 Line 3
   RUNG wire#powerrail
      Contact( "AlwaysTRUE" )
      wire#w1
      I_Contact( "BFT-61".state.Inloading )
      Contact( "General_Blend".Blend_Cluster1.CIP_Line3."CIP Request" )
      Coil( "General Buffer"."CIP Enable".Cluster1_Line3 )
   END_RUNG
   RUNG wire#w1
      Contact( "General Buffer"."CIP Enable".Cluster1_Line3 )
      Contact( "IO_Valve_Buffer_DB"."AV-62.06".FB_OPEN )
      Coil( "General Buffer"."CIP Line Open".Cluster1_Line3 )
   END_RUNG
   // the same network as SCL:
   "General Buffer"."CIP Enable".Cluster1_Line3 := "AlwaysTRUE" AND NOT "BFT-61".state.Inloading AND "General_Blend".Blend_Cluster1.CIP_Line3."CIP Request";
   "General Buffer"."CIP Line Open".Cluster1_Line3 := "AlwaysTRUE" AND "General Buffer"."CIP Enable".Cluster1_Line3 AND "IO_Valve_Buffer_DB"."AV-62.06".FB_OPEN;
END_REGION

REGION Network 33: CIP Enable and CIP Line Open for Blending Cluster Line 2 Line 1
   RUNG wire#powerrail
      Contact( "AlwaysTRUE" )
      wire#w1
      I_Contact( "BFT-64".state.Inloading )
      Contact( "General_Blend".Blend_Cluster2.CIP_Line1."CIP Request" )
      Coil( "General Buffer"."CIP Enable".Cluster2_Line1 )
   END_RUNG
   RUNG wire#w1
      Contact( "General Buffer"."CIP Enable".Cluster2_Line1 )
      Contact( "IO_Valve_Buffer_DB"."AV-64.06".FB_OPEN )
      Coil( "General Buffer"."CIP Line Open".Cluster2_Line1 )
   END_RUNG
   // the same network as SCL:
   "General Buffer"."CIP Enable".Cluster2_Line1 := "AlwaysTRUE" AND NOT "BFT-64".state.Inloading AND "General_Blend".Blend_Cluster2.CIP_Line1."CIP Request";
   "General Buffer"."CIP Line Open".Cluster2_Line1 := "AlwaysTRUE" AND "General Buffer"."CIP Enable".Cluster2_Line1 AND "IO_Valve_Buffer_DB"."AV-64.06".FB_OPEN;
END_REGION

REGION Network 34: CIP Enable and CIP Line Open for Blending Cluster Line 2 Line 2
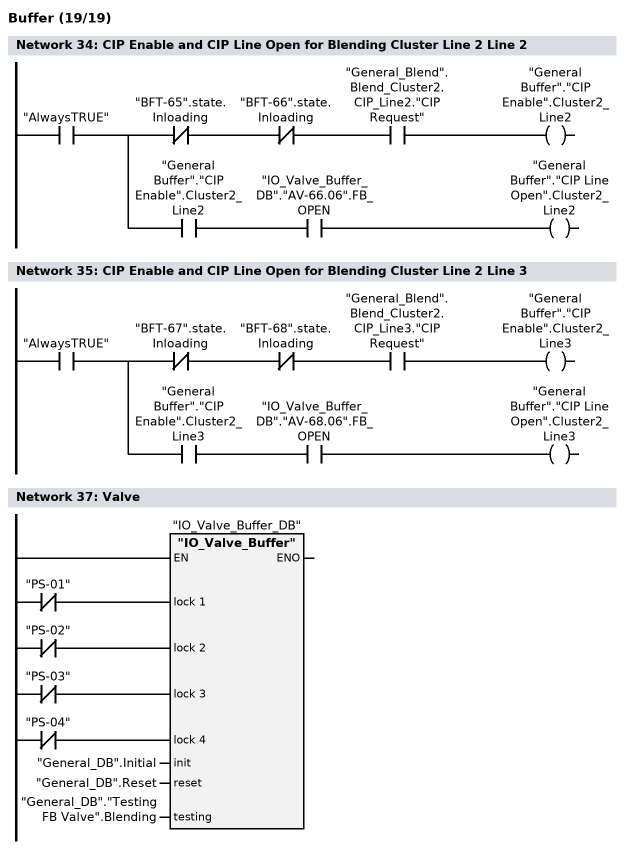
   RUNG wire#powerrail
      Contact( "AlwaysTRUE" )
      wire#w1
      I_Contact( "BFT-65".state.Inloading )
      I_Contact( "BFT-66".state.Inloading )
      Contact( "General_Blend".Blend_Cluster2.CIP_Line2."CIP Request" )
      Coil( "General Buffer"."CIP Enable".Cluster2_Line2 )
   END_RUNG
   RUNG wire#w1
      Contact( "General Buffer"."CIP Enable".Cluster2_Line2 )
      Contact( "IO_Valve_Buffer_DB"."AV-66.06".FB_OPEN )
      Coil( "General Buffer"."CIP Line Open".Cluster2_Line2 )
   END_RUNG
   // the same network as SCL:
   "General Buffer"."CIP Enable".Cluster2_Line2 := "AlwaysTRUE" AND NOT "BFT-65".state.Inloading AND NOT "BFT-66".state.Inloading AND "General_Blend".Blend_Cluster2.CIP_Line2."CIP Request";
   "General Buffer"."CIP Line Open".Cluster2_Line2 := "AlwaysTRUE" AND "General Buffer"."CIP Enable".Cluster2_Line2 AND "IO_Valve_Buffer_DB"."AV-66.06".FB_OPEN;
END_REGION

REGION Network 35: CIP Enable and CIP Line Open for Blending Cluster Line 2 Line 3
   RUNG wire#powerrail
      Contact( "AlwaysTRUE" )
      wire#w1
      I_Contact( "BFT-67".state.Inloading )
      I_Contact( "BFT-68".state.Inloading )
      Contact( "General_Blend".Blend_Cluster2.CIP_Line3."CIP Request" )
      Coil( "General Buffer"."CIP Enable".Cluster2_Line3 )
   END_RUNG
   RUNG wire#w1
      Contact( "General Buffer"."CIP Enable".Cluster2_Line3 )
      Contact( "IO_Valve_Buffer_DB"."AV-68.06".FB_OPEN )
      Coil( "General Buffer"."CIP Line Open".Cluster2_Line3 )
   END_RUNG
   // the same network as SCL:
   "General Buffer"."CIP Enable".Cluster2_Line3 := "AlwaysTRUE" AND NOT "BFT-67".state.Inloading AND NOT "BFT-68".state.Inloading AND "General_Blend".Blend_Cluster2.CIP_Line3."CIP Request";
   "General Buffer"."CIP Line Open".Cluster2_Line3 := "AlwaysTRUE" AND "General Buffer"."CIP Enable".Cluster2_Line3 AND "IO_Valve_Buffer_DB"."AV-68.06".FB_OPEN;
END_REGION

REGION Network 37: Valve
   RUNG wire#powerrail
      "IO_Valve_Buffer_DB"("lock 1" := wire#w1, "lock 2" := wire#w2, "lock 3" := wire#w3, "lock 4" := wire#w4, init := "General_DB".Initial, reset := "General_DB".Reset, testing := "General_DB"."Testing FB Valve".Blending)
   END_RUNG
   RUNG wire#powerrail
      I_Contact( "PS-01" )
   END_RUNG wire#w1
   RUNG wire#powerrail
      I_Contact( "PS-02" )
   END_RUNG wire#w2
   RUNG wire#powerrail
      I_Contact( "PS-03" )
   END_RUNG wire#w3
   RUNG wire#powerrail
      I_Contact( "PS-04" )
   END_RUNG wire#w4
   // the same network as SCL:
   "IO_Valve_Buffer_DB"("lock 1" := NOT "PS-01",   // "IO_Valve_Buffer"
                        "lock 2" := NOT "PS-02",
                        "lock 3" := NOT "PS-03",
                        "lock 4" := NOT "PS-04",
                        init := "General_DB".Initial,
                        reset := "General_DB".Reset,
                        testing := "General_DB"."Testing FB Valve".Blending);
END_REGION
END_FUNCTION
